//     Term 57 (AT2002-0250)/Term 58 (AT2002-5250)/FB Inputs/Value Channel 14 <-> Data Pointer/RawPositionValues[13]
//     Term 57 (AT2002-0250)/Term 58 (AT2002-5250)/FB Inputs/Value Channel 15 <-> Data Pointer/RawPositionValues[14]
//     Term 57 (AT2002-0250)/Term 58 (AT2002-5250)/FB Inputs/Value Channel 16 <-> Data Pointer/RawPositionValues[15]
//     Term 57 (AT2002-0250)/Term 58 (AT2002-5250)/FB Inputs/Value Channel 17 <-> Data Pointer/RawPositionValues[16]
//     Term 57 (AT2002-0250)/Term 58 (AT2002-5250)/FB Inputs/Value Channel 18 <-> Data Pointer/RawPositionValues[17]
//     Term 57 (AT2002-0250)/Term 58 (AT2002-5250)/FB Inputs/Value Channel 19 <-> Data Pointer/RawPositionValues[18]
//     Term 57 (AT2002-0250)/Term 58 (AT2002-5250)/FB Inputs/Value Channel 20 <-> Data Pointer/RawPositionValues[19]
//     Term 57 (AT2002-0250)/Term 58 (AT2002-5250)/FB Inputs/Value Channel 21 <-> Data Pointer/RawPositionValues[20]
//     Term 57 (AT2002-0250)/Term 58 (AT2002-5250)/FB Inputs/Value Channel 22 <-> Data Pointer/RawPositionValues[21]
//     Term 57 (AT2002-0250)/Term 58 (AT2002-5250)/FB Inputs/Value Channel 23 <-> Data Pointer/RawPositionValues[22]
//     Term 57 (AT2002-0250)/Term 58 (AT2002-5250)/FB Inputs/Value Channel 24 <-> Data Pointer/RawPositionValues[23]
//     Term 57 (AT2002-0250)/Term 58 (AT2002-5250)/FB Inputs/Value Channel 25 <-> Data Pointer/RawPositionValues[24]
//     Term 57 (AT2002-0250)/Term 58 (AT2002-5250)/FB Inputs/Value Channel 26 <-> Data Pointer/RawPositionValues[25]
//     Term 57 (AT2002-0250)/Term 58 (AT2002-5250)/FB Inputs/Value Channel 27 <-> Data Pointer/RawPositionValues[26]
//     Term 57 (AT2002-0250)/Term 58 (AT2002-5250)/FB Inputs/Value Channel 28 <-> Data Pointer/RawPositionValues[27]
//     Term 57 (AT2002-0250)/Term 58 (AT2002-5250)/FB Inputs/Value Channel 29 <-> Data Pointer/RawPositionValues[28]
//     Term 57 (AT2002-0250)/Term 58 (AT2002-5250)/FB Inputs/Value Channel 30 <-> Data Pointer/RawPositionValues[29]
//     Term 57 (AT2002-0250)/Term 58 (AT2002-5250)/FB Inputs/Value Channel 31 <-> Data Pointer/RawPositionValues[30]
//     Term 57 (AT2002-0250)/Term 58 (AT2002-5250)/FB Inputs/Value Channel 32 <-> Data Pointer/RawPositionValues[31]
//   Device 30 <-> TcCOM Objects/XTS ProcessingUnit 1/Part 1/Module 45
//     Term 59 (AT2200-0500)/CC Inputs/Current actual value Ch.1 <-> Data Pointer/CurrentActualValues[0]
//     Term 59 (AT2200-0500)/CC Inputs/Current actual value Ch.10 <-> Data Pointer/CurrentActualValues[9]
//     Term 59 (AT2200-0500)/CC Inputs/Current actual value Ch.11 <-> Data Pointer/CurrentActualValues[10]
//     Term 59 (AT2200-0500)/CC Inputs/Current actual value Ch.12 <-> Data Pointer/CurrentActualValues[11]
//     Term 59 (AT2200-0500)/CC Inputs/Current actual value Ch.13 <-> Data Pointer/CurrentActualValues[12]
//     Term 59 (AT2200-0500)/CC Inputs/Current actual value Ch.14 <-> Data Pointer/CurrentActualValues[13]
//     Term 59 (AT2200-0500)/CC Inputs/Current actual value Ch.15 <-> Data Pointer/CurrentActualValues[14]
//     Term 59 (AT2200-0500)/CC Inputs/Current actual value Ch.16 <-> Data Pointer/CurrentActualValues[15]
//     Term 59 (AT2200-0500)/CC Inputs/Current actual value Ch.17 <-> Data Pointer/CurrentActualValues[16]
//     Term 59 (AT2200-0500)/CC Inputs/Current actual value Ch.18 <-> Data Pointer/CurrentActualValues[17]
//     Term 59 (AT2200-0500)/CC Inputs/Current actual value Ch.19 <-> Data Pointer/CurrentActualValues[18]
//     Term 59 (AT2200-0500)/CC Inputs/Current actual value Ch.2 <-> Data Pointer/CurrentActualValues[1]
//     Term 59 (AT2200-0500)/CC Inputs/Current actual value Ch.20 <-> Data Pointer/CurrentActualValues[19]
//     Term 59 (AT2200-0500)/CC Inputs/Current actual value Ch.21 <-> Data Pointer/CurrentActualValues[20]
//     Term 59 (AT2200-0500)/CC Inputs/Current actual value Ch.22 <-> Data Pointer/CurrentActualValues[21]
//     Term 59 (AT2200-0500)/CC Inputs/Current actual value Ch.23 <-> Data Pointer/CurrentActualValues[22]
//     Term 59 (AT2200-0500)/CC Inputs/Current actual value Ch.24 <-> Data Pointer/CurrentActualValues[23]
//     Term 59 (AT2200-0500)/CC Inputs/Current actual value Ch.25 <-> Data Pointer/CurrentActualValues[24]
//     Term 59 (AT2200-0500)/CC Inputs/Current actual value Ch.26 <-> Data Pointer/CurrentActualValues[25]
//     Term 59 (AT2200-0500)/CC Inputs/Current actual value Ch.27 <-> Data Pointer/CurrentActualValues[26]
//     Term 59 (AT2200-0500)/CC Inputs/Current actual value Ch.28 <-> Data Pointer/CurrentActualValues[27]
//     Term 59 (AT2200-0500)/CC Inputs/Current actual value Ch.29 <-> Data Pointer/CurrentActualValues[28]
//     Term 59 (AT2200-0500)/CC Inputs/Current actual value Ch.3 <-> Data Pointer/CurrentActualValues[2]
//     Term 59 (AT2200-0500)/CC Inputs/Current actual value Ch.30 <-> Data Pointer/CurrentActualValues[29]
//     Term 59 (AT2200-0500)/CC Inputs/Current actual value Ch.4 <-> Data Pointer/CurrentActualValues[3]
//     Term 59 (AT2200-0500)/CC Inputs/Current actual value Ch.5 <-> Data Pointer/CurrentActualValues[4]
//     Term 59 (AT2200-0500)/CC Inputs/Current actual value Ch.6 <-> Data Pointer/CurrentActualValues[5]
//     Term 59 (AT2200-0500)/CC Inputs/Current actual value Ch.7 <-> Data Pointer/CurrentActualValues[6]
//     Term 59 (AT2200-0500)/CC Inputs/Current actual value Ch.8 <-> Data Pointer/CurrentActualValues[7]
//     Term 59 (AT2200-0500)/CC Inputs/Current actual value Ch.9 <-> Data Pointer/CurrentActualValues[8]
//     Term 59 (AT2200-0500)/CC Inputs/Status <-> Data Pointer/Status
//     Term 59 (AT2200-0500)/CC Outputs/Control <-> Data Pointer/Control
//     Term 59 (AT2200-0500)/CC Outputs/Current setpoint value Ch.1 <-> Data Pointer/CurrentSetpointValues[0]
//     Term 59 (AT2200-0500)/CC Outputs/Current setpoint value Ch.10 <-> Data Pointer/CurrentSetpointValues[9]
//     Term 59 (AT2200-0500)/CC Outputs/Current setpoint value Ch.11 <-> Data Pointer/CurrentSetpointValues[10]
//     Term 59 (AT2200-0500)/CC Outputs/Current setpoint value Ch.12 <-> Data Pointer/CurrentSetpointValues[11]
//     Term 59 (AT2200-0500)/CC Outputs/Current setpoint value Ch.13 <-> Data Pointer/CurrentSetpointValues[12]
//     Term 59 (AT2200-0500)/CC Outputs/Current setpoint value Ch.14 <-> Data Pointer/CurrentSetpointValues[13]
//     Term 59 (AT2200-0500)/CC Outputs/Current setpoint value Ch.15 <-> Data Pointer/CurrentSetpointValues[14]
//     Term 59 (AT2200-0500)/CC Outputs/Current setpoint value Ch.16 <-> Data Pointer/CurrentSetpointValues[15]
//     Term 59 (AT2200-0500)/CC Outputs/Current setpoint value Ch.17 <-> Data Pointer/CurrentSetpointValues[16]
//     Term 59 (AT2200-0500)/CC Outputs/Current setpoint value Ch.18 <-> Data Pointer/CurrentSetpointValues[17]
//     Term 59 (AT2200-0500)/CC Outputs/Current setpoint value Ch.19 <-> Data Pointer/CurrentSetpointValues[18]
//     Term 59 (AT2200-0500)/CC Outputs/Current setpoint value Ch.2 <-> Data Pointer/CurrentSetpointValues[1]
//     Term 59 (AT2200-0500)/CC Outputs/Current setpoint value Ch.20 <-> Data Pointer/CurrentSetpointValues[19]
//     Term 59 (AT2200-0500)/CC Outputs/Current setpoint value Ch.21 <-> Data Pointer/CurrentSetpointValues[20]
//     Term 59 (AT2200-0500)/CC Outputs/Current setpoint value Ch.22 <-> Data Pointer/CurrentSetpointValues[21]
//     Term 59 (AT2200-0500)/CC Outputs/Current setpoint value Ch.23 <-> Data Pointer/CurrentSetpointValues[22]
//     Term 59 (AT2200-0500)/CC Outputs/Current setpoint value Ch.24 <-> Data Pointer/CurrentSetpointValues[23]
//     Term 59 (AT2200-0500)/CC Outputs/Current setpoint value Ch.25 <-> Data Pointer/CurrentSetpointValues[24]
//     Term 59 (AT2200-0500)/CC Outputs/Current setpoint value Ch.26 <-> Data Pointer/CurrentSetpointValues[25]
//     Term 59 (AT2200-0500)/CC Outputs/Current setpoint value Ch.27 <-> Data Pointer/CurrentSetpointValues[26]
//     Term 59 (AT2200-0500)/CC Outputs/Current setpoint value Ch.28 <-> Data Pointer/CurrentSetpointValues[27]
//     Term 59 (AT2200-0500)/CC Outputs/Current setpoint value Ch.29 <-> Data Pointer/CurrentSetpointValues[28]
//     Term 59 (AT2200-0500)/CC Outputs/Current setpoint value Ch.3 <-> Data Pointer/CurrentSetpointValues[2]
//     Term 59 (AT2200-0500)/CC Outputs/Current setpoint value Ch.30 <-> Data Pointer/CurrentSetpointValues[29]
//     Term 59 (AT2200-0500)/CC Outputs/Current setpoint value Ch.4 <-> Data Pointer/CurrentSetpointValues[3]
//     Term 59 (AT2200-0500)/CC Outputs/Current setpoint value Ch.5 <-> Data Pointer/CurrentSetpointValues[4]
//     Term 59 (AT2200-0500)/CC Outputs/Current setpoint value Ch.6 <-> Data Pointer/CurrentSetpointValues[5]
//     Term 59 (AT2200-0500)/CC Outputs/Current setpoint value Ch.7 <-> Data Pointer/CurrentSetpointValues[6]
//     Term 59 (AT2200-0500)/CC Outputs/Current setpoint value Ch.8 <-> Data Pointer/CurrentSetpointValues[7]
//     Term 59 (AT2200-0500)/CC Outputs/Current setpoint value Ch.9 <-> Data Pointer/CurrentSetpointValues[8]
//     Term 59 (AT2200-0500)/LFB Inputs/BinaryData <-> Data Pointer/HallSensorValues
//   Device 30 <-> TcCOM Objects/XTS ProcessingUnit 1/Part 1/Module 46
//     Term 60 (AT2200-0500)/CC Inputs/Current actual value Ch.1 <-> Data Pointer/CurrentActualValues[0]
//     Term 60 (AT2200-0500)/CC Inputs/Current actual value Ch.10 <-> Data Pointer/CurrentActualValues[9]
//     Term 60 (AT2200-0500)/CC Inputs/Current actual value Ch.11 <-> Data Pointer/CurrentActualValues[10]
//     Term 60 (AT2200-0500)/CC Inputs/Current actual value Ch.12 <-> Data Pointer/CurrentActualValues[11]
//     Term 60 (AT2200-0500)/CC Inputs/Current actual value Ch.13 <-> Data Pointer/CurrentActualValues[12]
//     Term 60 (AT2200-0500)/CC Inputs/Current actual value Ch.14 <-> Data Pointer/CurrentActualValues[13]
//     Term 60 (AT2200-0500)/CC Inputs/Current actual value Ch.15 <-> Data Pointer/CurrentActualValues[14]
//     Term 60 (AT2200-0500)/CC Inputs/Current actual value Ch.16 <-> Data Pointer/CurrentActualValues[15]
//     Term 60 (AT2200-0500)/CC Inputs/Current actual value Ch.17 <-> Data Pointer/CurrentActualValues[16]
//     Term 60 (AT2200-0500)/CC Inputs/Current actual value Ch.18 <-> Data Pointer/CurrentActualValues[17]
//     Term 60 (AT2200-0500)/CC Inputs/Current actual value Ch.19 <-> Data Pointer/CurrentActualValues[18]
//     Term 60 (AT2200-0500)/CC Inputs/Current actual value Ch.2 <-> Data Pointer/CurrentActualValues[1]
//     Term 60 (AT2200-0500)/CC Inputs/Current actual value Ch.20 <-> Data Pointer/CurrentActualValues[19]
//     Term 60 (AT2200-0500)/CC Inputs/Current actual value Ch.21 <-> Data Pointer/CurrentActualValues[20]
//     Term 60 (AT2200-0500)/CC Inputs/Current actual value Ch.22 <-> Data Pointer/CurrentActualValues[21]
//     Term 60 (AT2200-0500)/CC Inputs/Current actual value Ch.23 <-> Data Pointer/CurrentActualValues[22]
//     Term 60 (AT2200-0500)/CC Inputs/Current actual value Ch.24 <-> Data Pointer/CurrentActualValues[23]
//     Term 60 (AT2200-0500)/CC Inputs/Current actual value Ch.25 <-> Data Pointer/CurrentActualValues[24]
//     Term 60 (AT2200-0500)/CC Inputs/Current actual value Ch.26 <-> Data Pointer/CurrentActualValues[25]
//     Term 60 (AT2200-0500)/CC Inputs/Current actual value Ch.27 <-> Data Pointer/CurrentActualValues[26]
//     Term 60 (AT2200-0500)/CC Inputs/Current actual value Ch.28 <-> Data Pointer/CurrentActualValues[27]
//     Term 60 (AT2200-0500)/CC Inputs/Current actual value Ch.29 <-> Data Pointer/CurrentActualValues[28]
//     Term 60 (AT2200-0500)/CC Inputs/Current actual value Ch.3 <-> Data Pointer/CurrentActualValues[2]
//     Term 60 (AT2200-0500)/CC Inputs/Current actual value Ch.30 <-> Data Pointer/CurrentActualValues[29]
//     Term 60 (AT2200-0500)/CC Inputs/Current actual value Ch.4 <-> Data Pointer/CurrentActualValues[3]
//     Term 60 (AT2200-0500)/CC Inputs/Current actual value Ch.5 <-> Data Pointer/CurrentActualValues[4]
//     Term 60 (AT2200-0500)/CC Inputs/Current actual value Ch.6 <-> Data Pointer/CurrentActualValues[5]
//     Term 60 (AT2200-0500)/CC Inputs/Current actual value Ch.7 <-> Data Pointer/CurrentActualValues[6]
//     Term 60 (AT2200-0500)/CC Inputs/Current actual value Ch.8 <-> Data Pointer/CurrentActualValues[7]
//     Term 60 (AT2200-0500)/CC Inputs/Current actual value Ch.9 <-> Data Pointer/CurrentActualValues[8]
//     Term 60 (AT2200-0500)/CC Inputs/Status <-> Data Pointer/Status
//     Term 60 (AT2200-0500)/CC Outputs/Control <-> Data Pointer/Control
//     Term 60 (AT2200-0500)/CC Outputs/Current setpoint value Ch.1 <-> Data Pointer/CurrentSetpointValues[0]
//     Term 60 (AT2200-0500)/CC Outputs/Current setpoint value Ch.10 <-> Data Pointer/CurrentSetpointValues[9]
//     Term 60 (AT2200-0500)/CC Outputs/Current setpoint value Ch.11 <-> Data Pointer/CurrentSetpointValues[10]
//     Term 60 (AT2200-0500)/CC Outputs/Current setpoint value Ch.12 <-> Data Pointer/CurrentSetpointValues[11]
//     Term 60 (AT2200-0500)/CC Outputs/Current setpoint value Ch.13 <-> Data Pointer/CurrentSetpointValues[12]
//     Term 60 (AT2200-0500)/CC Outputs/Current setpoint value Ch.14 <-> Data Pointer/CurrentSetpointValues[13]
//     Term 60 (AT2200-0500)/CC Outputs/Current setpoint value Ch.15 <-> Data Pointer/CurrentSetpointValues[14]
//     Term 60 (AT2200-0500)/CC Outputs/Current setpoint value Ch.16 <-> Data Pointer/CurrentSetpointValues[15]
//     Term 60 (AT2200-0500)/CC Outputs/Current setpoint value Ch.17 <-> Data Pointer/CurrentSetpointValues[16]
//     Term 60 (AT2200-0500)/CC Outputs/Current setpoint value Ch.18 <-> Data Pointer/CurrentSetpointValues[17]
//     Term 60 (AT2200-0500)/CC Outputs/Current setpoint value Ch.19 <-> Data Pointer/CurrentSetpointValues[18]
//     Term 60 (AT2200-0500)/CC Outputs/Current setpoint value Ch.2 <-> Data Pointer/CurrentSetpointValues[1]
//     Term 60 (AT2200-0500)/CC Outputs/Current setpoint value Ch.20 <-> Data Pointer/CurrentSetpointValues[19]
//     Term 60 (AT2200-0500)/CC Outputs/Current setpoint value Ch.21 <-> Data Pointer/CurrentSetpointValues[20]
//     Term 60 (AT2200-0500)/CC Outputs/Current setpoint value Ch.22 <-> Data Pointer/CurrentSetpointValues[21]
//     Term 60 (AT2200-0500)/CC Outputs/Current setpoint value Ch.23 <-> Data Pointer/CurrentSetpointValues[22]
//     Term 60 (AT2200-0500)/CC Outputs/Current setpoint value Ch.24 <-> Data Pointer/CurrentSetpointValues[23]
//     Term 60 (AT2200-0500)/CC Outputs/Current setpoint value Ch.25 <-> Data Pointer/CurrentSetpointValues[24]
//     Term 60 (AT2200-0500)/CC Outputs/Current setpoint value Ch.26 <-> Data Pointer/CurrentSetpointValues[25]
//     Term 60 (AT2200-0500)/CC Outputs/Current setpoint value Ch.27 <-> Data Pointer/CurrentSetpointValues[26]
//     Term 60 (AT2200-0500)/CC Outputs/Current setpoint value Ch.28 <-> Data Pointer/CurrentSetpointValues[27]
//     Term 60 (AT2200-0500)/CC Outputs/Current setpoint value Ch.29 <-> Data Pointer/CurrentSetpointValues[28]
//     Term 60 (AT2200-0500)/CC Outputs/Current setpoint value Ch.3 <-> Data Pointer/CurrentSetpointValues[2]
//     Term 60 (AT2200-0500)/CC Outputs/Current setpoint value Ch.30 <-> Data Pointer/CurrentSetpointValues[29]
//     Term 60 (AT2200-0500)/CC Outputs/Current setpoint value Ch.4 <-> Data Pointer/CurrentSetpointValues[3]
//     Term 60 (AT2200-0500)/CC Outputs/Current setpoint value Ch.5 <-> Data Pointer/CurrentSetpointValues[4]
//     Term 60 (AT2200-0500)/CC Outputs/Current setpoint value Ch.6 <-> Data Pointer/CurrentSetpointValues[5]
//     Term 60 (AT2200-0500)/CC Outputs/Current setpoint value Ch.7 <-> Data Pointer/CurrentSetpointValues[6]
//     Term 60 (AT2200-0500)/CC Outputs/Current setpoint value Ch.8 <-> Data Pointer/CurrentSetpointValues[7]
//     Term 60 (AT2200-0500)/CC Outputs/Current setpoint value Ch.9 <-> Data Pointer/CurrentSetpointValues[8]
//     Term 60 (AT2200-0500)/LFB Inputs/BinaryData <-> Data Pointer/HallSensorValues
//   Device 31 <-> TcCOM Objects/XTS ProcessingUnit 1/Part 1/Module 47
//     Term 61 (AT2202-0500)/CC Inputs/Current actual value Ch.1 <-> Data Pointer/CurrentActualValues[0]
//     Term 61 (AT2202-0500)/CC Inputs/Current actual value Ch.10 <-> Data Pointer/CurrentActualValues[9]
//     Term 61 (AT2202-0500)/CC Inputs/Current actual value Ch.11 <-> Data Pointer/CurrentActualValues[10]
//     Term 61 (AT2202-0500)/CC Inputs/Current actual value Ch.12 <-> Data Pointer/CurrentActualValues[11]
//     Term 61 (AT2202-0500)/CC Inputs/Current actual value Ch.13 <-> Data Pointer/CurrentActualValues[12]
//     Term 61 (AT2202-0500)/CC Inputs/Current actual value Ch.14 <-> Data Pointer/CurrentActualValues[13]
//     Term 61 (AT2202-0500)/CC Inputs/Current actual value Ch.15 <-> Data Pointer/CurrentActualValues[14]
//     Term 61 (AT2202-0500)/CC Inputs/Current actual value Ch.16 <-> Data Pointer/CurrentActualValues[15]
//     Term 61 (AT2202-0500)/CC Inputs/Current actual value Ch.17 <-> Data Pointer/CurrentActualValues[16]
//     Term 61 (AT2202-0500)/CC Inputs/Current actual value Ch.18 <-> Data Pointer/CurrentActualValues[17]
//     Term 61 (AT2202-0500)/CC Inputs/Current actual value Ch.19 <-> Data Pointer/CurrentActualValues[18]
//     Term 61 (AT2202-0500)/CC Inputs/Current actual value Ch.2 <-> Data Pointer/CurrentActualValues[1]
//     Term 61 (AT2202-0500)/CC Inputs/Current actual value Ch.20 <-> Data Pointer/CurrentActualValues[19]
//     Term 61 (AT2202-0500)/CC Inputs/Current actual value Ch.21 <-> Data Pointer/CurrentActualValues[20]
//     Term 61 (AT2202-0500)/CC Inputs/Current actual value Ch.22 <-> Data Pointer/CurrentActualValues[21]
//     Term 61 (AT2202-0500)/CC Inputs/Current actual value Ch.23 <-> Data Pointer/CurrentActualValues[22]
//     Term 61 (AT2202-0500)/CC Inputs/Current actual value Ch.24 <-> Data Pointer/CurrentActualValues[23]
//     Term 61 (AT2202-0500)/CC Inputs/Current actual value Ch.25 <-> Data Pointer/CurrentActualValues[24]
//     Term 61 (AT2202-0500)/CC Inputs/Current actual value Ch.26 <-> Data Pointer/CurrentActualValues[25]
//     Term 61 (AT2202-0500)/CC Inputs/Current actual value Ch.27 <-> Data Pointer/CurrentActualValues[26]
//     Term 61 (AT2202-0500)/CC Inputs/Current actual value Ch.28 <-> Data Pointer/CurrentActualValues[27]
//     Term 61 (AT2202-0500)/CC Inputs/Current actual value Ch.29 <-> Data Pointer/CurrentActualValues[28]
//     Term 61 (AT2202-0500)/CC Inputs/Current actual value Ch.3 <-> Data Pointer/CurrentActualValues[2]
//     Term 61 (AT2202-0500)/CC Inputs/Current actual value Ch.30 <-> Data Pointer/CurrentActualValues[29]
//     Term 61 (AT2202-0500)/CC Inputs/Current actual value Ch.4 <-> Data Pointer/CurrentActualValues[3]
//     Term 61 (AT2202-0500)/CC Inputs/Current actual value Ch.5 <-> Data Pointer/CurrentActualValues[4]
//     Term 61 (AT2202-0500)/CC Inputs/Current actual value Ch.6 <-> Data Pointer/CurrentActualValues[5]
//     Term 61 (AT2202-0500)/CC Inputs/Current actual value Ch.7 <-> Data Pointer/CurrentActualValues[6]
//     Term 61 (AT2202-0500)/CC Inputs/Current actual value Ch.8 <-> Data Pointer/CurrentActualValues[7]
//     Term 61 (AT2202-0500)/CC Inputs/Current actual value Ch.9 <-> Data Pointer/CurrentActualValues[8]
//     Term 61 (AT2202-0500)/CC Inputs/Status <-> Data Pointer/Status
//     Term 61 (AT2202-0500)/CC Outputs/Control <-> Data Pointer/Control
//     Term 61 (AT2202-0500)/CC Outputs/Current setpoint value Ch.1 <-> Data Pointer/CurrentSetpointValues[0]
//     Term 61 (AT2202-0500)/CC Outputs/Current setpoint value Ch.10 <-> Data Pointer/CurrentSetpointValues[9]
//     Term 61 (AT2202-0500)/CC Outputs/Current setpoint value Ch.11 <-> Data Pointer/CurrentSetpointValues[10]
//     Term 61 (AT2202-0500)/CC Outputs/Current setpoint value Ch.12 <-> Data Pointer/CurrentSetpointValues[11]
//     Term 61 (AT2202-0500)/CC Outputs/Current setpoint value Ch.13 <-> Data Pointer/CurrentSetpointValues[12]
//     Term 61 (AT2202-0500)/CC Outputs/Current setpoint value Ch.14 <-> Data Pointer/CurrentSetpointValues[13]
//     Term 61 (AT2202-0500)/CC Outputs/Current setpoint value Ch.15 <-> Data Pointer/CurrentSetpointValues[14]
//     Term 61 (AT2202-0500)/CC Outputs/Current setpoint value Ch.16 <-> Data Pointer/CurrentSetpointValues[15]
//     Term 61 (AT2202-0500)/CC Outputs/Current setpoint value Ch.17 <-> Data Pointer/CurrentSetpointValues[16]
//     Term 61 (AT2202-0500)/CC Outputs/Current setpoint value Ch.18 <-> Data Pointer/CurrentSetpointValues[17]
//     Term 61 (AT2202-0500)/CC Outputs/Current setpoint value Ch.19 <-> Data Pointer/CurrentSetpointValues[18]
//     Term 61 (AT2202-0500)/CC Outputs/Current setpoint value Ch.2 <-> Data Pointer/CurrentSetpointValues[1]
//     Term 61 (AT2202-0500)/CC Outputs/Current setpoint value Ch.20 <-> Data Pointer/CurrentSetpointValues[19]
//     Term 61 (AT2202-0500)/CC Outputs/Current setpoint value Ch.21 <-> Data Pointer/CurrentSetpointValues[20]
//     Term 61 (AT2202-0500)/CC Outputs/Current setpoint value Ch.22 <-> Data Pointer/CurrentSetpointValues[21]
//     Term 61 (AT2202-0500)/CC Outputs/Current setpoint value Ch.23 <-> Data Pointer/CurrentSetpointValues[22]
//     Term 61 (AT2202-0500)/CC Outputs/Current setpoint value Ch.24 <-> Data Pointer/CurrentSetpointValues[23]
//     Term 61 (AT2202-0500)/CC Outputs/Current setpoint value Ch.25 <-> Data Pointer/CurrentSetpointValues[24]
//     Term 61 (AT2202-0500)/CC Outputs/Current setpoint value Ch.26 <-> Data Pointer/CurrentSetpointValues[25]
//     Term 61 (AT2202-0500)/CC Outputs/Current setpoint value Ch.27 <-> Data Pointer/CurrentSetpointValues[26]
//     Term 61 (AT2202-0500)/CC Outputs/Current setpoint value Ch.28 <-> Data Pointer/CurrentSetpointValues[27]
//     Term 61 (AT2202-0500)/CC Outputs/Current setpoint value Ch.29 <-> Data Pointer/CurrentSetpointValues[28]
//     Term 61 (AT2202-0500)/CC Outputs/Current setpoint value Ch.3 <-> Data Pointer/CurrentSetpointValues[2]
//     Term 61 (AT2202-0500)/CC Outputs/Current setpoint value Ch.30 <-> Data Pointer/CurrentSetpointValues[29]
//     Term 61 (AT2202-0500)/CC Outputs/Current setpoint value Ch.4 <-> Data Pointer/CurrentSetpointValues[3]
//     Term 61 (AT2202-0500)/CC Outputs/Current setpoint value Ch.5 <-> Data Pointer/CurrentSetpointValues[4]
//     Term 61 (AT2202-0500)/CC Outputs/Current setpoint value Ch.6 <-> Data Pointer/CurrentSetpointValues[5]
//     Term 61 (AT2202-0500)/CC Outputs/Current setpoint value Ch.7 <-> Data Pointer/CurrentSetpointValues[6]
//     Term 61 (AT2202-0500)/CC Outputs/Current setpoint value Ch.8 <-> Data Pointer/CurrentSetpointValues[7]
//     Term 61 (AT2202-0500)/CC Outputs/Current setpoint value Ch.9 <-> Data Pointer/CurrentSetpointValues[8]
//     Term 61 (AT2202-0500)/LFB Inputs/BinaryData <-> Data Pointer/HallSensorValues
//   Device 31 <-> TcCOM Objects/XTS ProcessingUnit 1/Part 1/Module 48
//     Term 62 (AT2200-0500)/CC Inputs/Current actual value Ch.1 <-> Data Pointer/CurrentActualValues[0]
//     Term 62 (AT2200-0500)/CC Inputs/Current actual value Ch.10 <-> Data Pointer/CurrentActualValues[9]
//     Term 62 (AT2200-0500)/CC Inputs/Current actual value Ch.11 <-> Data Pointer/CurrentActualValues[10]
//     Term 62 (AT2200-0500)/CC Inputs/Current actual value Ch.12 <-> Data Pointer/CurrentActualValues[11]
//     Term 62 (AT2200-0500)/CC Inputs/Current actual value Ch.13 <-> Data Pointer/CurrentActualValues[12]
//     Term 62 (AT2200-0500)/CC Inputs/Current actual value Ch.14 <-> Data Pointer/CurrentActualValues[13]
//     Term 62 (AT2200-0500)/CC Inputs/Current actual value Ch.15 <-> Data Pointer/CurrentActualValues[14]
//     Term 62 (AT2200-0500)/CC Inputs/Current actual value Ch.16 <-> Data Pointer/CurrentActualValues[15]
//     Term 62 (AT2200-0500)/CC Inputs/Current actual value Ch.17 <-> Data Pointer/CurrentActualValues[16]
//     Term 62 (AT2200-0500)/CC Inputs/Current actual value Ch.18 <-> Data Pointer/CurrentActualValues[17]
//     Term 62 (AT2200-0500)/CC Inputs/Current actual value Ch.19 <-> Data Pointer/CurrentActualValues[18]
//     Term 62 (AT2200-0500)/CC Inputs/Current actual value Ch.2 <-> Data Pointer/CurrentActualValues[1]
//     Term 62 (AT2200-0500)/CC Inputs/Current actual value Ch.20 <-> Data Pointer/CurrentActualValues[19]
//     Term 62 (AT2200-0500)/CC Inputs/Current actual value Ch.21 <-> Data Pointer/CurrentActualValues[20]
//     Term 62 (AT2200-0500)/CC Inputs/Current actual value Ch.22 <-> Data Pointer/CurrentActualValues[21]
//     Term 62 (AT2200-0500)/CC Inputs/Current actual value Ch.23 <-> Data Pointer/CurrentActualValues[22]
//     Term 62 (AT2200-0500)/CC Inputs/Current actual value Ch.24 <-> Data Pointer/CurrentActualValues[23]
//     Term 62 (AT2200-0500)/CC Inputs/Current actual value Ch.25 <-> Data Pointer/CurrentActualValues[24]
//     Term 62 (AT2200-0500)/CC Inputs/Current actual value Ch.26 <-> Data Pointer/CurrentActualValues[25]
//     Term 62 (AT2200-0500)/CC Inputs/Current actual value Ch.27 <-> Data Pointer/CurrentActualValues[26]
//     Term 62 (AT2200-0500)/CC Inputs/Current actual value Ch.28 <-> Data Pointer/CurrentActualValues[27]
//     Term 62 (AT2200-0500)/CC Inputs/Current actual value Ch.29 <-> Data Pointer/CurrentActualValues[28]
//     Term 62 (AT2200-0500)/CC Inputs/Current actual value Ch.3 <-> Data Pointer/CurrentActualValues[2]
//     Term 62 (AT2200-0500)/CC Inputs/Current actual value Ch.30 <-> Data Pointer/CurrentActualValues[29]
//     Term 62 (AT2200-0500)/CC Inputs/Current actual value Ch.4 <-> Data Pointer/CurrentActualValues[3]
//     Term 62 (AT2200-0500)/CC Inputs/Current actual value Ch.5 <-> Data Pointer/CurrentActualValues[4]
//     Term 62 (AT2200-0500)/CC Inputs/Current actual value Ch.6 <-> Data Pointer/CurrentActualValues[5]
//     Term 62 (AT2200-0500)/CC Inputs/Current actual value Ch.7 <-> Data Pointer/CurrentActualValues[6]
//     Term 62 (AT2200-0500)/CC Inputs/Current actual value Ch.8 <-> Data Pointer/CurrentActualValues[7]
//     Term 62 (AT2200-0500)/CC Inputs/Current actual value Ch.9 <-> Data Pointer/CurrentActualValues[8]
//     Term 62 (AT2200-0500)/CC Inputs/Status <-> Data Pointer/Status
//     Term 62 (AT2200-0500)/CC Outputs/Control <-> Data Pointer/Control
//     Term 62 (AT2200-0500)/CC Outputs/Current setpoint value Ch.1 <-> Data Pointer/CurrentSetpointValues[0]
//     Term 62 (AT2200-0500)/CC Outputs/Current setpoint value Ch.10 <-> Data Pointer/CurrentSetpointValues[9]
//     Term 62 (AT2200-0500)/CC Outputs/Current setpoint value Ch.11 <-> Data Pointer/CurrentSetpointValues[10]
//     Term 62 (AT2200-0500)/CC Outputs/Current setpoint value Ch.12 <-> Data Pointer/CurrentSetpointValues[11]
//     Term 62 (AT2200-0500)/CC Outputs/Current setpoint value Ch.13 <-> Data Pointer/CurrentSetpointValues[12]
//     Term 62 (AT2200-0500)/CC Outputs/Current setpoint value Ch.14 <-> Data Pointer/CurrentSetpointValues[13]
//     Term 62 (AT2200-0500)/CC Outputs/Current setpoint value Ch.15 <-> Data Pointer/CurrentSetpointValues[14]
//     Term 62 (AT2200-0500)/CC Outputs/Current setpoint value Ch.16 <-> Data Pointer/CurrentSetpointValues[15]
//     Term 62 (AT2200-0500)/CC Outputs/Current setpoint value Ch.17 <-> Data Pointer/CurrentSetpointValues[16]
//     Term 62 (AT2200-0500)/CC Outputs/Current setpoint value Ch.18 <-> Data Pointer/CurrentSetpointValues[17]
//     Term 62 (AT2200-0500)/CC Outputs/Current setpoint value Ch.19 <-> Data Pointer/CurrentSetpointValues[18]
//     Term 62 (AT2200-0500)/CC Outputs/Current setpoint value Ch.2 <-> Data Pointer/CurrentSetpointValues[1]
//     Term 62 (AT2200-0500)/CC Outputs/Current setpoint value Ch.20 <-> Data Pointer/CurrentSetpointValues[19]
//     Term 62 (AT2200-0500)/CC Outputs/Current setpoint value Ch.21 <-> Data Pointer/CurrentSetpointValues[20]
//     Term 62 (AT2200-0500)/CC Outputs/Current setpoint value Ch.22 <-> Data Pointer/CurrentSetpointValues[21]
//     Term 62 (AT2200-0500)/CC Outputs/Current setpoint value Ch.23 <-> Data Pointer/CurrentSetpointValues[22]
//     Term 62 (AT2200-0500)/CC Outputs/Current setpoint value Ch.24 <-> Data Pointer/CurrentSetpointValues[23]
//     Term 62 (AT2200-0500)/CC Outputs/Current setpoint value Ch.25 <-> Data Pointer/CurrentSetpointValues[24]
//     Term 62 (AT2200-0500)/CC Outputs/Current setpoint value Ch.26 <-> Data Pointer/CurrentSetpointValues[25]
//     Term 62 (AT2200-0500)/CC Outputs/Current setpoint value Ch.27 <-> Data Pointer/CurrentSetpointValues[26]
//     Term 62 (AT2200-0500)/CC Outputs/Current setpoint value Ch.28 <-> Data Pointer/CurrentSetpointValues[27]
//     Term 62 (AT2200-0500)/CC Outputs/Current setpoint value Ch.29 <-> Data Pointer/CurrentSetpointValues[28]
//     Term 62 (AT2200-0500)/CC Outputs/Current setpoint value Ch.3 <-> Data Pointer/CurrentSetpointValues[2]
//     Term 62 (AT2200-0500)/CC Outputs/Current setpoint value Ch.30 <-> Data Pointer/CurrentSetpointValues[29]
//     Term 62 (AT2200-0500)/CC Outputs/Current setpoint value Ch.4 <-> Data Pointer/CurrentSetpointValues[3]
//     Term 62 (AT2200-0500)/CC Outputs/Current setpoint value Ch.5 <-> Data Pointer/CurrentSetpointValues[4]
//     Term 62 (AT2200-0500)/CC Outputs/Current setpoint value Ch.6 <-> Data Pointer/CurrentSetpointValues[5]
//     Term 62 (AT2200-0500)/CC Outputs/Current setpoint value Ch.7 <-> Data Pointer/CurrentSetpointValues[6]
//     Term 62 (AT2200-0500)/CC Outputs/Current setpoint value Ch.8 <-> Data Pointer/CurrentSetpointValues[7]
//     Term 62 (AT2200-0500)/CC Outputs/Current setpoint value Ch.9 <-> Data Pointer/CurrentSetpointValues[8]
//     Term 62 (AT2200-0500)/LFB Inputs/BinaryData <-> Data Pointer/HallSensorValues
//   Device 31 <-> TcCOM Objects/XTS ProcessingUnit 1/Part 1/Module 49
//     Term 63 (AT2000-0250)/CC Inputs/Current actual value Ch.1 <-> Data Pointer/CurrentActualValues[0]
//     Term 63 (AT2000-0250)/CC Inputs/Current actual value Ch.10 <-> Data Pointer/CurrentActualValues[9]
//     Term 63 (AT2000-0250)/CC Inputs/Current actual value Ch.11 <-> Data Pointer/CurrentActualValues[10]
//     Term 63 (AT2000-0250)/CC Inputs/Current actual value Ch.12 <-> Data Pointer/CurrentActualValues[11]
//     Term 63 (AT2000-0250)/CC Inputs/Current actual value Ch.13 <-> Data Pointer/CurrentActualValues[12]
//     Term 63 (AT2000-0250)/CC Inputs/Current actual value Ch.14 <-> Data Pointer/CurrentActualValues[13]
//     Term 63 (AT2000-0250)/CC Inputs/Current actual value Ch.15 <-> Data Pointer/CurrentActualValues[14]
//     Term 63 (AT2000-0250)/CC Inputs/Current actual value Ch.2 <-> Data Pointer/CurrentActualValues[1]
//     Term 63 (AT2000-0250)/CC Inputs/Current actual value Ch.3 <-> Data Pointer/CurrentActualValues[2]
//     Term 63 (AT2000-0250)/CC Inputs/Current actual value Ch.4 <-> Data Pointer/CurrentActualValues[3]
//     Term 63 (AT2000-0250)/CC Inputs/Current actual value Ch.5 <-> Data Pointer/CurrentActualValues[4]
//     Term 63 (AT2000-0250)/CC Inputs/Current actual value Ch.6 <-> Data Pointer/CurrentActualValues[5]
//     Term 63 (AT2000-0250)/CC Inputs/Current actual value Ch.7 <-> Data Pointer/CurrentActualValues[6]
//     Term 63 (AT2000-0250)/CC Inputs/Current actual value Ch.8 <-> Data Pointer/CurrentActualValues[7]
//     Term 63 (AT2000-0250)/CC Inputs/Current actual value Ch.9 <-> Data Pointer/CurrentActualValues[8]
//     Term 63 (AT2000-0250)/CC Inputs/Status <-> Data Pointer/Status
//     Term 63 (AT2000-0250)/CC Outputs/Control <-> Data Pointer/Control
//     Term 63 (AT2000-0250)/CC Outputs/Current setpoint value Ch.1 <-> Data Pointer/CurrentSetpointValues[0]
//     Term 63 (AT2000-0250)/CC Outputs/Current setpoint value Ch.10 <-> Data Pointer/CurrentSetpointValues[9]
//     Term 63 (AT2000-0250)/CC Outputs/Current setpoint value Ch.11 <-> Data Pointer/CurrentSetpointValues[10]
//     Term 63 (AT2000-0250)/CC Outputs/Current setpoint value Ch.12 <-> Data Pointer/CurrentSetpointValues[11]
//     Term 63 (AT2000-0250)/CC Outputs/Current setpoint value Ch.13 <-> Data Pointer/CurrentSetpointValues[12]
//     Term 63 (AT2000-0250)/CC Outputs/Current setpoint value Ch.14 <-> Data Pointer/CurrentSetpointValues[13]
//     Term 63 (AT2000-0250)/CC Outputs/Current setpoint value Ch.15 <-> Data Pointer/CurrentSetpointValues[14]
//     Term 63 (AT2000-0250)/CC Outputs/Current setpoint value Ch.2 <-> Data Pointer/CurrentSetpointValues[1]
//     Term 63 (AT2000-0250)/CC Outputs/Current setpoint value Ch.3 <-> Data Pointer/CurrentSetpointValues[2]
//     Term 63 (AT2000-0250)/CC Outputs/Current setpoint value Ch.4 <-> Data Pointer/CurrentSetpointValues[3]
//     Term 63 (AT2000-0250)/CC Outputs/Current setpoint value Ch.5 <-> Data Pointer/CurrentSetpointValues[4]
//     Term 63 (AT2000-0250)/CC Outputs/Current setpoint value Ch.6 <-> Data Pointer/CurrentSetpointValues[5]
//     Term 63 (AT2000-0250)/CC Outputs/Current setpoint value Ch.7 <-> Data Pointer/CurrentSetpointValues[6]
//     Term 63 (AT2000-0250)/CC Outputs/Current setpoint value Ch.8 <-> Data Pointer/CurrentSetpointValues[7]
//     Term 63 (AT2000-0250)/CC Outputs/Current setpoint value Ch.9 <-> Data Pointer/CurrentSetpointValues[8]
//     Term 63 (AT2000-0250)/Term 64 (AT2000-5250)/FB Inputs/Value Channel 01 <-> Data Pointer/RawPositionValues[0]
//     Term 63 (AT2000-0250)/Term 64 (AT2000-5250)/FB Inputs/Value Channel 02 <-> Data Pointer/RawPositionValues[1]
//     Term 63 (AT2000-0250)/Term 64 (AT2000-5250)/FB Inputs/Value Channel 03 <-> Data Pointer/RawPositionValues[2]
//     Term 63 (AT2000-0250)/Term 64 (AT2000-5250)/FB Inputs/Value Channel 04 <-> Data Pointer/RawPositionValues[3]
//     Term 63 (AT2000-0250)/Term 64 (AT2000-5250)/FB Inputs/Value Channel 05 <-> Data Pointer/RawPositionValues[4]
//     Term 63 (AT2000-0250)/Term 64 (AT2000-5250)/FB Inputs/Value Channel 06 <-> Data Pointer/RawPositionValues[5]
//     Term 63 (AT2000-0250)/Term 64 (AT2000-5250)/FB Inputs/Value Channel 07 <-> Data Pointer/RawPositionValues[6]
//     Term 63 (AT2000-0250)/Term 64 (AT2000-5250)/FB Inputs/Value Channel 08 <-> Data Pointer/RawPositionValues[7]
//     Term 63 (AT2000-0250)/Term 64 (AT2000-5250)/FB Inputs/Value Channel 09 <-> Data Pointer/RawPositionValues[8]
//     Term 63 (AT2000-0250)/Term 64 (AT2000-5250)/FB Inputs/Value Channel 10 <-> Data Pointer/RawPositionValues[9]
//     Term 63 (AT2000-0250)/Term 64 (AT2000-5250)/FB Inputs/Value Channel 11 <-> Data Pointer/RawPositionValues[10]
//     Term 63 (AT2000-0250)/Term 64 (AT2000-5250)/FB Inputs/Value Channel 12 <-> Data Pointer/RawPositionValues[11]
//     Term 63 (AT2000-0250)/Term 64 (AT2000-5250)/FB Inputs/Value Channel 13 <-> Data Pointer/RawPositionValues[12]
//     Term 63 (AT2000-0250)/Term 64 (AT2000-5250)/FB Inputs/Value Channel 14 <-> Data Pointer/RawPositionValues[13]
//     Term 63 (AT2000-0250)/Term 64 (AT2000-5250)/FB Inputs/Value Channel 15 <-> Data Pointer/RawPositionValues[14]
//     Term 63 (AT2000-0250)/Term 64 (AT2000-5250)/FB Inputs/Value Channel 16 <-> Data Pointer/RawPositionValues[15]
//     Term 63 (AT2000-0250)/Term 64 (AT2000-5250)/FB Inputs/Value Channel 17 <-> Data Pointer/RawPositionValues[16]
//     Term 63 (AT2000-0250)/Term 64 (AT2000-5250)/FB Inputs/Value Channel 18 <-> Data Pointer/RawPositionValues[17]
//     Term 63 (AT2000-0250)/Term 64 (AT2000-5250)/FB Inputs/Value Channel 19 <-> Data Pointer/RawPositionValues[18]
//     Term 63 (AT2000-0250)/Term 64 (AT2000-5250)/FB Inputs/Value Channel 20 <-> Data Pointer/RawPositionValues[19]
//     Term 63 (AT2000-0250)/Term 64 (AT2000-5250)/FB Inputs/Value Channel 21 <-> Data Pointer/RawPositionValues[20]
//     Term 63 (AT2000-0250)/Term 64 (AT2000-5250)/FB Inputs/Value Channel 22 <-> Data Pointer/RawPositionValues[21]
//     Term 63 (AT2000-0250)/Term 64 (AT2000-5250)/FB Inputs/Value Channel 23 <-> Data Pointer/RawPositionValues[22]
//     Term 63 (AT2000-0250)/Term 64 (AT2000-5250)/FB Inputs/Value Channel 24 <-> Data Pointer/RawPositionValues[23]
//     Term 63 (AT2000-0250)/Term 64 (AT2000-5250)/FB Inputs/Value Channel 25 <-> Data Pointer/RawPositionValues[24]
//     Term 63 (AT2000-0250)/Term 64 (AT2000-5250)/FB Inputs/Value Channel 26 <-> Data Pointer/RawPositionValues[25]
//     Term 63 (AT2000-0250)/Term 64 (AT2000-5250)/FB Inputs/Value Channel 27 <-> Data Pointer/RawPositionValues[26]
//     Term 63 (AT2000-0250)/Term 64 (AT2000-5250)/FB Inputs/Value Channel 28 <-> Data Pointer/RawPositionValues[27]
//     Term 63 (AT2000-0250)/Term 64 (AT2000-5250)/FB Inputs/Value Channel 29 <-> Data Pointer/RawPositionValues[28]
//     Term 63 (AT2000-0250)/Term 64 (AT2000-5250)/FB Inputs/Value Channel 30 <-> Data Pointer/RawPositionValues[29]
//     Term 63 (AT2000-0250)/Term 64 (AT2000-5250)/FB Inputs/Value Channel 31 <-> Data Pointer/RawPositionValues[30]
//     Term 63 (AT2000-0250)/Term 64 (AT2000-5250)/FB Inputs/Value Channel 32 <-> Data Pointer/RawPositionValues[31]
//   Device 32 <-> TcCOM Objects/XTS ProcessingUnit 1/Part 1/Module 50
//     Term 65 (AT2002-0250)/CC Inputs/Current actual value Ch.1 <-> Data Pointer/CurrentActualValues[0]
//     Term 65 (AT2002-0250)/CC Inputs/Current actual value Ch.10 <-> Data Pointer/CurrentActualValues[9]
//     Term 65 (AT2002-0250)/CC Inputs/Current actual value Ch.11 <-> Data Pointer/CurrentActualValues[10]
//     Term 65 (AT2002-0250)/CC Inputs/Current actual value Ch.12 <-> Data Pointer/CurrentActualValues[11]
//     Term 65 (AT2002-0250)/CC Inputs/Current actual value Ch.13 <-> Data Pointer/CurrentActualValues[12]
//     Term 65 (AT2002-0250)/CC Inputs/Current actual value Ch.14 <-> Data Pointer/CurrentActualValues[13]
//     Term 65 (AT2002-0250)/CC Inputs/Current actual value Ch.15 <-> Data Pointer/CurrentActualValues[14]
//     Term 65 (AT2002-0250)/CC Inputs/Current actual value Ch.2 <-> Data Pointer/CurrentActualValues[1]
//     Term 65 (AT2002-0250)/CC Inputs/Current actual value Ch.3 <-> Data Pointer/CurrentActualValues[2]
//     Term 65 (AT2002-0250)/CC Inputs/Current actual value Ch.4 <-> Data Pointer/CurrentActualValues[3]
//     Term 65 (AT2002-0250)/CC Inputs/Current actual value Ch.5 <-> Data Pointer/CurrentActualValues[4]
//     Term 65 (AT2002-0250)/CC Inputs/Current actual value Ch.6 <-> Data Pointer/CurrentActualValues[5]
//     Term 65 (AT2002-0250)/CC Inputs/Current actual value Ch.7 <-> Data Pointer/CurrentActualValues[6]
//     Term 65 (AT2002-0250)/CC Inputs/Current actual value Ch.8 <-> Data Pointer/CurrentActualValues[7]
//     Term 65 (AT2002-0250)/CC Inputs/Current actual value Ch.9 <-> Data Pointer/CurrentActualValues[8]
//     Term 65 (AT2002-0250)/CC Inputs/Status <-> Data Pointer/Status
//     Term 65 (AT2002-0250)/CC Outputs/Control <-> Data Pointer/Control
//     Term 65 (AT2002-0250)/CC Outputs/Current setpoint value Ch.1 <-> Data Pointer/CurrentSetpointValues[0]
//     Term 65 (AT2002-0250)/CC Outputs/Current setpoint value Ch.10 <-> Data Pointer/CurrentSetpointValues[9]
//     Term 65 (AT2002-0250)/CC Outputs/Current setpoint value Ch.11 <-> Data Pointer/CurrentSetpointValues[10]
//     Term 65 (AT2002-0250)/CC Outputs/Current setpoint value Ch.12 <-> Data Pointer/CurrentSetpointValues[11]
//     Term 65 (AT2002-0250)/CC Outputs/Current setpoint value Ch.13 <-> Data Pointer/CurrentSetpointValues[12]
//     Term 65 (AT2002-0250)/CC Outputs/Current setpoint value Ch.14 <-> Data Pointer/CurrentSetpointValues[13]
//     Term 65 (AT2002-0250)/CC Outputs/Current setpoint value Ch.15 <-> Data Pointer/CurrentSetpointValues[14]
//     Term 65 (AT2002-0250)/CC Outputs/Current setpoint value Ch.2 <-> Data Pointer/CurrentSetpointValues[1]
//     Term 65 (AT2002-0250)/CC Outputs/Current setpoint value Ch.3 <-> Data Pointer/CurrentSetpointValues[2]
//     Term 65 (AT2002-0250)/CC Outputs/Current setpoint value Ch.4 <-> Data Pointer/CurrentSetpointValues[3]
//     Term 65 (AT2002-0250)/CC Outputs/Current setpoint value Ch.5 <-> Data Pointer/CurrentSetpointValues[4]
//     Term 65 (AT2002-0250)/CC Outputs/Current setpoint value Ch.6 <-> Data Pointer/CurrentSetpointValues[5]
//     Term 65 (AT2002-0250)/CC Outputs/Current setpoint value Ch.7 <-> Data Pointer/CurrentSetpointValues[6]
//     Term 65 (AT2002-0250)/CC Outputs/Current setpoint value Ch.8 <-> Data Pointer/CurrentSetpointValues[7]
//     Term 65 (AT2002-0250)/CC Outputs/Current setpoint value Ch.9 <-> Data Pointer/CurrentSetpointValues[8]
//     Term 65 (AT2002-0250)/Term 66 (AT2002-5250)/FB Inputs/Value Channel 01 <-> Data Pointer/RawPositionValues[0]
//     Term 65 (AT2002-0250)/Term 66 (AT2002-5250)/FB Inputs/Value Channel 02 <-> Data Pointer/RawPositionValues[1]
//     Term 65 (AT2002-0250)/Term 66 (AT2002-5250)/FB Inputs/Value Channel 03 <-> Data Pointer/RawPositionValues[2]
//     Term 65 (AT2002-0250)/Term 66 (AT2002-5250)/FB Inputs/Value Channel 04 <-> Data Pointer/RawPositionValues[3]
//     Term 65 (AT2002-0250)/Term 66 (AT2002-5250)/FB Inputs/Value Channel 05 <-> Data Pointer/RawPositionValues[4]
//     Term 65 (AT2002-0250)/Term 66 (AT2002-5250)/FB Inputs/Value Channel 06 <-> Data Pointer/RawPositionValues[5]
//     Term 65 (AT2002-0250)/Term 66 (AT2002-5250)/FB Inputs/Value Channel 07 <-> Data Pointer/RawPositionValues[6]
//     Term 65 (AT2002-0250)/Term 66 (AT2002-5250)/FB Inputs/Value Channel 08 <-> Data Pointer/RawPositionValues[7]
//     Term 65 (AT2002-0250)/Term 66 (AT2002-5250)/FB Inputs/Value Channel 09 <-> Data Pointer/RawPositionValues[8]
//     Term 65 (AT2002-0250)/Term 66 (AT2002-5250)/FB Inputs/Value Channel 10 <-> Data Pointer/RawPositionValues[9]
//     Term 65 (AT2002-0250)/Term 66 (AT2002-5250)/FB Inputs/Value Channel 11 <-> Data Pointer/RawPositionValues[10]
//     Term 65 (AT2002-0250)/Term 66 (AT2002-5250)/FB Inputs/Value Channel 12 <-> Data Pointer/RawPositionValues[11]
//     Term 65 (AT2002-0250)/Term 66 (AT2002-5250)/FB Inputs/Value Channel 13 <-> Data Pointer/RawPositionValues[12]
//     Term 65 (AT2002-0250)/Term 66 (AT2002-5250)/FB Inputs/Value Channel 14 <-> Data Pointer/RawPositionValues[13]
//     Term 65 (AT2002-0250)/Term 66 (AT2002-5250)/FB Inputs/Value Channel 15 <-> Data Pointer/RawPositionValues[14]
//     Term 65 (AT2002-0250)/Term 66 (AT2002-5250)/FB Inputs/Value Channel 16 <-> Data Pointer/RawPositionValues[15]
//     Term 65 (AT2002-0250)/Term 66 (AT2002-5250)/FB Inputs/Value Channel 17 <-> Data Pointer/RawPositionValues[16]
//     Term 65 (AT2002-0250)/Term 66 (AT2002-5250)/FB Inputs/Value Channel 18 <-> Data Pointer/RawPositionValues[17]
//     Term 65 (AT2002-0250)/Term 66 (AT2002-5250)/FB Inputs/Value Channel 19 <-> Data Pointer/RawPositionValues[18]
//     Term 65 (AT2002-0250)/Term 66 (AT2002-5250)/FB Inputs/Value Channel 20 <-> Data Pointer/RawPositionValues[19]
//     Term 65 (AT2002-0250)/Term 66 (AT2002-5250)/FB Inputs/Value Channel 21 <-> Data Pointer/RawPositionValues[20]
//     Term 65 (AT2002-0250)/Term 66 (AT2002-5250)/FB Inputs/Value Channel 22 <-> Data Pointer/RawPositionValues[21]
//     Term 65 (AT2002-0250)/Term 66 (AT2002-5250)/FB Inputs/Value Channel 23 <-> Data Pointer/RawPositionValues[22]
//     Term 65 (AT2002-0250)/Term 66 (AT2002-5250)/FB Inputs/Value Channel 24 <-> Data Pointer/RawPositionValues[23]
//     Term 65 (AT2002-0250)/Term 66 (AT2002-5250)/FB Inputs/Value Channel 25 <-> Data Pointer/RawPositionValues[24]
//     Term 65 (AT2002-0250)/Term 66 (AT2002-5250)/FB Inputs/Value Channel 26 <-> Data Pointer/RawPositionValues[25]
//     Term 65 (AT2002-0250)/Term 66 (AT2002-5250)/FB Inputs/Value Channel 27 <-> Data Pointer/RawPositionValues[26]
//     Term 65 (AT2002-0250)/Term 66 (AT2002-5250)/FB Inputs/Value Channel 28 <-> Data Pointer/RawPositionValues[27]
//     Term 65 (AT2002-0250)/Term 66 (AT2002-5250)/FB Inputs/Value Channel 29 <-> Data Pointer/RawPositionValues[28]
//     Term 65 (AT2002-0250)/Term 66 (AT2002-5250)/FB Inputs/Value Channel 30 <-> Data Pointer/RawPositionValues[29]
//     Term 65 (AT2002-0250)/Term 66 (AT2002-5250)/FB Inputs/Value Channel 31 <-> Data Pointer/RawPositionValues[30]
//     Term 65 (AT2002-0250)/Term 66 (AT2002-5250)/FB Inputs/Value Channel 32 <-> Data Pointer/RawPositionValues[31]
//   Device 32 <-> TcCOM Objects/XTS ProcessingUnit 1/Part 1/Module 51
//     Term 67 (AT2200-0500)/CC Inputs/Current actual value Ch.1 <-> Data Pointer/CurrentActualValues[0]
//     Term 67 (AT2200-0500)/CC Inputs/Current actual value Ch.10 <-> Data Pointer/CurrentActualValues[9]
//     Term 67 (AT2200-0500)/CC Inputs/Current actual value Ch.11 <-> Data Pointer/CurrentActualValues[10]
//     Term 67 (AT2200-0500)/CC Inputs/Current actual value Ch.12 <-> Data Pointer/CurrentActualValues[11]
//     Term 67 (AT2200-0500)/CC Inputs/Current actual value Ch.13 <-> Data Pointer/CurrentActualValues[12]
//     Term 67 (AT2200-0500)/CC Inputs/Current actual value Ch.14 <-> Data Pointer/CurrentActualValues[13]
//     Term 67 (AT2200-0500)/CC Inputs/Current actual value Ch.15 <-> Data Pointer/CurrentActualValues[14]
//     Term 67 (AT2200-0500)/CC Inputs/Current actual value Ch.16 <-> Data Pointer/CurrentActualValues[15]
//     Term 67 (AT2200-0500)/CC Inputs/Current actual value Ch.17 <-> Data Pointer/CurrentActualValues[16]
//     Term 67 (AT2200-0500)/CC Inputs/Current actual value Ch.18 <-> Data Pointer/CurrentActualValues[17]
//     Term 67 (AT2200-0500)/CC Inputs/Current actual value Ch.19 <-> Data Pointer/CurrentActualValues[18]
//     Term 67 (AT2200-0500)/CC Inputs/Current actual value Ch.2 <-> Data Pointer/CurrentActualValues[1]
//     Term 67 (AT2200-0500)/CC Inputs/Current actual value Ch.20 <-> Data Pointer/CurrentActualValues[19]
//     Term 67 (AT2200-0500)/CC Inputs/Current actual value Ch.21 <-> Data Pointer/CurrentActualValues[20]
//     Term 67 (AT2200-0500)/CC Inputs/Current actual value Ch.22 <-> Data Pointer/CurrentActualValues[21]
//     Term 67 (AT2200-0500)/CC Inputs/Current actual value Ch.23 <-> Data Pointer/CurrentActualValues[22]
//     Term 67 (AT2200-0500)/CC Inputs/Current actual value Ch.24 <-> Data Pointer/CurrentActualValues[23]
//     Term 67 (AT2200-0500)/CC Inputs/Current actual value Ch.25 <-> Data Pointer/CurrentActualValues[24]
//     Term 67 (AT2200-0500)/CC Inputs/Current actual value Ch.26 <-> Data Pointer/CurrentActualValues[25]
//     Term 67 (AT2200-0500)/CC Inputs/Current actual value Ch.27 <-> Data Pointer/CurrentActualValues[26]
//     Term 67 (AT2200-0500)/CC Inputs/Current actual value Ch.28 <-> Data Pointer/CurrentActualValues[27]
//     Term 67 (AT2200-0500)/CC Inputs/Current actual value Ch.29 <-> Data Pointer/CurrentActualValues[28]
//     Term 67 (AT2200-0500)/CC Inputs/Current actual value Ch.3 <-> Data Pointer/CurrentActualValues[2]
//     Term 67 (AT2200-0500)/CC Inputs/Current actual value Ch.30 <-> Data Pointer/CurrentActualValues[29]
//     Term 67 (AT2200-0500)/CC Inputs/Current actual value Ch.4 <-> Data Pointer/CurrentActualValues[3]
//     Term 67 (AT2200-0500)/CC Inputs/Current actual value Ch.5 <-> Data Pointer/CurrentActualValues[4]
//     Term 67 (AT2200-0500)/CC Inputs/Current actual value Ch.6 <-> Data Pointer/CurrentActualValues[5]
//     Term 67 (AT2200-0500)/CC Inputs/Current actual value Ch.7 <-> Data Pointer/CurrentActualValues[6]
//     Term 67 (AT2200-0500)/CC Inputs/Current actual value Ch.8 <-> Data Pointer/CurrentActualValues[7]
//     Term 67 (AT2200-0500)/CC Inputs/Current actual value Ch.9 <-> Data Pointer/CurrentActualValues[8]
//     Term 67 (AT2200-0500)/CC Inputs/Status <-> Data Pointer/Status
//     Term 67 (AT2200-0500)/CC Outputs/Control <-> Data Pointer/Control
//     Term 67 (AT2200-0500)/CC Outputs/Current setpoint value Ch.1 <-> Data Pointer/CurrentSetpointValues[0]
//     Term 67 (AT2200-0500)/CC Outputs/Current setpoint value Ch.10 <-> Data Pointer/CurrentSetpointValues[9]
//     Term 67 (AT2200-0500)/CC Outputs/Current setpoint value Ch.11 <-> Data Pointer/CurrentSetpointValues[10]
//     Term 67 (AT2200-0500)/CC Outputs/Current setpoint value Ch.12 <-> Data Pointer/CurrentSetpointValues[11]
//     Term 67 (AT2200-0500)/CC Outputs/Current setpoint value Ch.13 <-> Data Pointer/CurrentSetpointValues[12]
//     Term 67 (AT2200-0500)/CC Outputs/Current setpoint value Ch.14 <-> Data Pointer/CurrentSetpointValues[13]
//     Term 67 (AT2200-0500)/CC Outputs/Current setpoint value Ch.15 <-> Data Pointer/CurrentSetpointValues[14]
//     Term 67 (AT2200-0500)/CC Outputs/Current setpoint value Ch.16 <-> Data Pointer/CurrentSetpointValues[15]
//     Term 67 (AT2200-0500)/CC Outputs/Current setpoint value Ch.17 <-> Data Pointer/CurrentSetpointValues[16]
//     Term 67 (AT2200-0500)/CC Outputs/Current setpoint value Ch.18 <-> Data Pointer/CurrentSetpointValues[17]
//     Term 67 (AT2200-0500)/CC Outputs/Current setpoint value Ch.19 <-> Data Pointer/CurrentSetpointValues[18]
//     Term 67 (AT2200-0500)/CC Outputs/Current setpoint value Ch.2 <-> Data Pointer/CurrentSetpointValues[1]
//     Term 67 (AT2200-0500)/CC Outputs/Current setpoint value Ch.20 <-> Data Pointer/CurrentSetpointValues[19]
//     Term 67 (AT2200-0500)/CC Outputs/Current setpoint value Ch.21 <-> Data Pointer/CurrentSetpointValues[20]
//     Term 67 (AT2200-0500)/CC Outputs/Current setpoint value Ch.22 <-> Data Pointer/CurrentSetpointValues[21]
//     Term 67 (AT2200-0500)/CC Outputs/Current setpoint value Ch.23 <-> Data Pointer/CurrentSetpointValues[22]
//     Term 67 (AT2200-0500)/CC Outputs/Current setpoint value Ch.24 <-> Data Pointer/CurrentSetpointValues[23]
//     Term 67 (AT2200-0500)/CC Outputs/Current setpoint value Ch.25 <-> Data Pointer/CurrentSetpointValues[24]
//     Term 67 (AT2200-0500)/CC Outputs/Current setpoint value Ch.26 <-> Data Pointer/CurrentSetpointValues[25]
//     Term 67 (AT2200-0500)/CC Outputs/Current setpoint value Ch.27 <-> Data Pointer/CurrentSetpointValues[26]
//     Term 67 (AT2200-0500)/CC Outputs/Current setpoint value Ch.28 <-> Data Pointer/CurrentSetpointValues[27]
//     Term 67 (AT2200-0500)/CC Outputs/Current setpoint value Ch.29 <-> Data Pointer/CurrentSetpointValues[28]
//     Term 67 (AT2200-0500)/CC Outputs/Current setpoint value Ch.3 <-> Data Pointer/CurrentSetpointValues[2]
//     Term 67 (AT2200-0500)/CC Outputs/Current setpoint value Ch.30 <-> Data Pointer/CurrentSetpointValues[29]
//     Term 67 (AT2200-0500)/CC Outputs/Current setpoint value Ch.4 <-> Data Pointer/CurrentSetpointValues[3]
//     Term 67 (AT2200-0500)/CC Outputs/Current setpoint value Ch.5 <-> Data Pointer/CurrentSetpointValues[4]
//     Term 67 (AT2200-0500)/CC Outputs/Current setpoint value Ch.6 <-> Data Pointer/CurrentSetpointValues[5]
//     Term 67 (AT2200-0500)/CC Outputs/Current setpoint value Ch.7 <-> Data Pointer/CurrentSetpointValues[6]
//     Term 67 (AT2200-0500)/CC Outputs/Current setpoint value Ch.8 <-> Data Pointer/CurrentSetpointValues[7]
//     Term 67 (AT2200-0500)/CC Outputs/Current setpoint value Ch.9 <-> Data Pointer/CurrentSetpointValues[8]
//     Term 67 (AT2200-0500)/LFB Inputs/BinaryData <-> Data Pointer/HallSensorValues
//   Device 32 <-> TcCOM Objects/XTS ProcessingUnit 1/Part 1/Module 52
//     Term 68 (AT2200-0500)/CC Inputs/Current actual value Ch.1 <-> Data Pointer/CurrentActualValues[0]
//     Term 68 (AT2200-0500)/CC Inputs/Current actual value Ch.10 <-> Data Pointer/CurrentActualValues[9]
//     Term 68 (AT2200-0500)/CC Inputs/Current actual value Ch.11 <-> Data Pointer/CurrentActualValues[10]
//     Term 68 (AT2200-0500)/CC Inputs/Current actual value Ch.12 <-> Data Pointer/CurrentActualValues[11]
//     Term 68 (AT2200-0500)/CC Inputs/Current actual value Ch.13 <-> Data Pointer/CurrentActualValues[12]
//     Term 68 (AT2200-0500)/CC Inputs/Current actual value Ch.14 <-> Data Pointer/CurrentActualValues[13]
//     Term 68 (AT2200-0500)/CC Inputs/Current actual value Ch.15 <-> Data Pointer/CurrentActualValues[14]
//     Term 68 (AT2200-0500)/CC Inputs/Current actual value Ch.16 <-> Data Pointer/CurrentActualValues[15]
//     Term 68 (AT2200-0500)/CC Inputs/Current actual value Ch.17 <-> Data Pointer/CurrentActualValues[16]
//     Term 68 (AT2200-0500)/CC Inputs/Current actual value Ch.18 <-> Data Pointer/CurrentActualValues[17]
//     Term 68 (AT2200-0500)/CC Inputs/Current actual value Ch.19 <-> Data Pointer/CurrentActualValues[18]
//     Term 68 (AT2200-0500)/CC Inputs/Current actual value Ch.2 <-> Data Pointer/CurrentActualValues[1]
//     Term 68 (AT2200-0500)/CC Inputs/Current actual value Ch.20 <-> Data Pointer/CurrentActualValues[19]
//     Term 68 (AT2200-0500)/CC Inputs/Current actual value Ch.21 <-> Data Pointer/CurrentActualValues[20]
//     Term 68 (AT2200-0500)/CC Inputs/Current actual value Ch.22 <-> Data Pointer/CurrentActualValues[21]
//     Term 68 (AT2200-0500)/CC Inputs/Current actual value Ch.23 <-> Data Pointer/CurrentActualValues[22]
//     Term 68 (AT2200-0500)/CC Inputs/Current actual value Ch.24 <-> Data Pointer/CurrentActualValues[23]
//     Term 68 (AT2200-0500)/CC Inputs/Current actual value Ch.25 <-> Data Pointer/CurrentActualValues[24]
//     Term 68 (AT2200-0500)/CC Inputs/Current actual value Ch.26 <-> Data Pointer/CurrentActualValues[25]
//     Term 68 (AT2200-0500)/CC Inputs/Current actual value Ch.27 <-> Data Pointer/CurrentActualValues[26]
//     Term 68 (AT2200-0500)/CC Inputs/Current actual value Ch.28 <-> Data Pointer/CurrentActualValues[27]
//     Term 68 (AT2200-0500)/CC Inputs/Current actual value Ch.29 <-> Data Pointer/CurrentActualValues[28]
//     Term 68 (AT2200-0500)/CC Inputs/Current actual value Ch.3 <-> Data Pointer/CurrentActualValues[2]
//     Term 68 (AT2200-0500)/CC Inputs/Current actual value Ch.30 <-> Data Pointer/CurrentActualValues[29]
//     Term 68 (AT2200-0500)/CC Inputs/Current actual value Ch.4 <-> Data Pointer/CurrentActualValues[3]
//     Term 68 (AT2200-0500)/CC Inputs/Current actual value Ch.5 <-> Data Pointer/CurrentActualValues[4]
//     Term 68 (AT2200-0500)/CC Inputs/Current actual value Ch.6 <-> Data Pointer/CurrentActualValues[5]
//     Term 68 (AT2200-0500)/CC Inputs/Current actual value Ch.7 <-> Data Pointer/CurrentActualValues[6]
//     Term 68 (AT2200-0500)/CC Inputs/Current actual value Ch.8 <-> Data Pointer/CurrentActualValues[7]
//     Term 68 (AT2200-0500)/CC Inputs/Current actual value Ch.9 <-> Data Pointer/CurrentActualValues[8]
//     Term 68 (AT2200-0500)/CC Inputs/Status <-> Data Pointer/Status
//     Term 68 (AT2200-0500)/CC Outputs/Control <-> Data Pointer/Control
//     Term 68 (AT2200-0500)/CC Outputs/Current setpoint value Ch.1 <-> Data Pointer/CurrentSetpointValues[0]
//     Term 68 (AT2200-0500)/CC Outputs/Current setpoint value Ch.10 <-> Data Pointer/CurrentSetpointValues[9]
//     Term 68 (AT2200-0500)/CC Outputs/Current setpoint value Ch.11 <-> Data Pointer/CurrentSetpointValues[10]
//     Term 68 (AT2200-0500)/CC Outputs/Current setpoint value Ch.12 <-> Data Pointer/CurrentSetpointValues[11]
//     Term 68 (AT2200-0500)/CC Outputs/Current setpoint value Ch.13 <-> Data Pointer/CurrentSetpointValues[12]
//     Term 68 (AT2200-0500)/CC Outputs/Current setpoint value Ch.14 <-> Data Pointer/CurrentSetpointValues[13]
//     Term 68 (AT2200-0500)/CC Outputs/Current setpoint value Ch.15 <-> Data Pointer/CurrentSetpointValues[14]
//     Term 68 (AT2200-0500)/CC Outputs/Current setpoint value Ch.16 <-> Data Pointer/CurrentSetpointValues[15]
//     Term 68 (AT2200-0500)/CC Outputs/Current setpoint value Ch.17 <-> Data Pointer/CurrentSetpointValues[16]
//     Term 68 (AT2200-0500)/CC Outputs/Current setpoint value Ch.18 <-> Data Pointer/CurrentSetpointValues[17]
//     Term 68 (AT2200-0500)/CC Outputs/Current setpoint value Ch.19 <-> Data Pointer/CurrentSetpointValues[18]
//     Term 68 (AT2200-0500)/CC Outputs/Current setpoint value Ch.2 <-> Data Pointer/CurrentSetpointValues[1]
//     Term 68 (AT2200-0500)/CC Outputs/Current setpoint value Ch.20 <-> Data Pointer/CurrentSetpointValues[19]
//     Term 68 (AT2200-0500)/CC Outputs/Current setpoint value Ch.21 <-> Data Pointer/CurrentSetpointValues[20]
//     Term 68 (AT2200-0500)/CC Outputs/Current setpoint value Ch.22 <-> Data Pointer/CurrentSetpointValues[21]
//     Term 68 (AT2200-0500)/CC Outputs/Current setpoint value Ch.23 <-> Data Pointer/CurrentSetpointValues[22]
//     Term 68 (AT2200-0500)/CC Outputs/Current setpoint value Ch.24 <-> Data Pointer/CurrentSetpointValues[23]
//     Term 68 (AT2200-0500)/CC Outputs/Current setpoint value Ch.25 <-> Data Pointer/CurrentSetpointValues[24]
//     Term 68 (AT2200-0500)/CC Outputs/Current setpoint value Ch.26 <-> Data Pointer/CurrentSetpointValues[25]
//     Term 68 (AT2200-0500)/CC Outputs/Current setpoint value Ch.27 <-> Data Pointer/CurrentSetpointValues[26]
//     Term 68 (AT2200-0500)/CC Outputs/Current setpoint value Ch.28 <-> Data Pointer/CurrentSetpointValues[27]
//     Term 68 (AT2200-0500)/CC Outputs/Current setpoint value Ch.29 <-> Data Pointer/CurrentSetpointValues[28]
//     Term 68 (AT2200-0500)/CC Outputs/Current setpoint value Ch.3 <-> Data Pointer/CurrentSetpointValues[2]
//     Term 68 (AT2200-0500)/CC Outputs/Current setpoint value Ch.30 <-> Data Pointer/CurrentSetpointValues[29]
//     Term 68 (AT2200-0500)/CC Outputs/Current setpoint value Ch.4 <-> Data Pointer/CurrentSetpointValues[3]
//     Term 68 (AT2200-0500)/CC Outputs/Current setpoint value Ch.5 <-> Data Pointer/CurrentSetpointValues[4]
//     Term 68 (AT2200-0500)/CC Outputs/Current setpoint value Ch.6 <-> Data Pointer/CurrentSetpointValues[5]
//     Term 68 (AT2200-0500)/CC Outputs/Current setpoint value Ch.7 <-> Data Pointer/CurrentSetpointValues[6]
//     Term 68 (AT2200-0500)/CC Outputs/Current setpoint value Ch.8 <-> Data Pointer/CurrentSetpointValues[7]
//     Term 68 (AT2200-0500)/CC Outputs/Current setpoint value Ch.9 <-> Data Pointer/CurrentSetpointValues[8]
//     Term 68 (AT2200-0500)/LFB Inputs/BinaryData <-> Data Pointer/HallSensorValues
//   Device 33 <-> TcCOM Objects/XTS ProcessingUnit 1/Part 1/Module 53
//     Term 69 (AT2042-0250)/CC Inputs/Current actual value Ch.1 <-> Data Pointer/CurrentActualValues[0]
//     Term 69 (AT2042-0250)/CC Inputs/Current actual value Ch.10 <-> Data Pointer/CurrentActualValues[9]
//     Term 69 (AT2042-0250)/CC Inputs/Current actual value Ch.11 <-> Data Pointer/CurrentActualValues[10]
//     Term 69 (AT2042-0250)/CC Inputs/Current actual value Ch.12 <-> Data Pointer/CurrentActualValues[11]
//     Term 69 (AT2042-0250)/CC Inputs/Current actual value Ch.13 <-> Data Pointer/CurrentActualValues[12]
//     Term 69 (AT2042-0250)/CC Inputs/Current actual value Ch.14 <-> Data Pointer/CurrentActualValues[13]
//     Term 69 (AT2042-0250)/CC Inputs/Current actual value Ch.15 <-> Data Pointer/CurrentActualValues[14]
//     Term 69 (AT2042-0250)/CC Inputs/Current actual value Ch.2 <-> Data Pointer/CurrentActualValues[1]
//     Term 69 (AT2042-0250)/CC Inputs/Current actual value Ch.3 <-> Data Pointer/CurrentActualValues[2]
//     Term 69 (AT2042-0250)/CC Inputs/Current actual value Ch.4 <-> Data Pointer/CurrentActualValues[3]
//     Term 69 (AT2042-0250)/CC Inputs/Current actual value Ch.5 <-> Data Pointer/CurrentActualValues[4]
//     Term 69 (AT2042-0250)/CC Inputs/Current actual value Ch.6 <-> Data Pointer/CurrentActualValues[5]
//     Term 69 (AT2042-0250)/CC Inputs/Current actual value Ch.7 <-> Data Pointer/CurrentActualValues[6]
//     Term 69 (AT2042-0250)/CC Inputs/Current actual value Ch.8 <-> Data Pointer/CurrentActualValues[7]
//     Term 69 (AT2042-0250)/CC Inputs/Current actual value Ch.9 <-> Data Pointer/CurrentActualValues[8]
//     Term 69 (AT2042-0250)/CC Inputs/Status <-> Data Pointer/Status
//     Term 69 (AT2042-0250)/CC Outputs/Control <-> Data Pointer/Control
//     Term 69 (AT2042-0250)/CC Outputs/Current setpoint value Ch.1 <-> Data Pointer/CurrentSetpointValues[0]
//     Term 69 (AT2042-0250)/CC Outputs/Current setpoint value Ch.10 <-> Data Pointer/CurrentSetpointValues[9]
//     Term 69 (AT2042-0250)/CC Outputs/Current setpoint value Ch.11 <-> Data Pointer/CurrentSetpointValues[10]
//     Term 69 (AT2042-0250)/CC Outputs/Current setpoint value Ch.12 <-> Data Pointer/CurrentSetpointValues[11]
//     Term 69 (AT2042-0250)/CC Outputs/Current setpoint value Ch.13 <-> Data Pointer/CurrentSetpointValues[12]
//     Term 69 (AT2042-0250)/CC Outputs/Current setpoint value Ch.14 <-> Data Pointer/CurrentSetpointValues[13]
//     Term 69 (AT2042-0250)/CC Outputs/Current setpoint value Ch.15 <-> Data Pointer/CurrentSetpointValues[14]
//     Term 69 (AT2042-0250)/CC Outputs/Current setpoint value Ch.2 <-> Data Pointer/CurrentSetpointValues[1]
//     Term 69 (AT2042-0250)/CC Outputs/Current setpoint value Ch.3 <-> Data Pointer/CurrentSetpointValues[2]
//     Term 69 (AT2042-0250)/CC Outputs/Current setpoint value Ch.4 <-> Data Pointer/CurrentSetpointValues[3]
//     Term 69 (AT2042-0250)/CC Outputs/Current setpoint value Ch.5 <-> Data Pointer/CurrentSetpointValues[4]
//     Term 69 (AT2042-0250)/CC Outputs/Current setpoint value Ch.6 <-> Data Pointer/CurrentSetpointValues[5]
//     Term 69 (AT2042-0250)/CC Outputs/Current setpoint value Ch.7 <-> Data Pointer/CurrentSetpointValues[6]
//     Term 69 (AT2042-0250)/CC Outputs/Current setpoint value Ch.8 <-> Data Pointer/CurrentSetpointValues[7]
//     Term 69 (AT2042-0250)/CC Outputs/Current setpoint value Ch.9 <-> Data Pointer/CurrentSetpointValues[8]
//     Term 69 (AT2042-0250)/Term 70 (AT2042-5250)/FB Inputs/Value Channel 01 <-> Data Pointer/RawPositionValues[0]
//     Term 69 (AT2042-0250)/Term 70 (AT2042-5250)/FB Inputs/Value Channel 02 <-> Data Pointer/RawPositionValues[1]
//     Term 69 (AT2042-0250)/Term 70 (AT2042-5250)/FB Inputs/Value Channel 03 <-> Data Pointer/RawPositionValues[2]
//     Term 69 (AT2042-0250)/Term 70 (AT2042-5250)/FB Inputs/Value Channel 04 <-> Data Pointer/RawPositionValues[3]
//     Term 69 (AT2042-0250)/Term 70 (AT2042-5250)/FB Inputs/Value Channel 05 <-> Data Pointer/RawPositionValues[4]
//     Term 69 (AT2042-0250)/Term 70 (AT2042-5250)/FB Inputs/Value Channel 06 <-> Data Pointer/RawPositionValues[5]
//     Term 69 (AT2042-0250)/Term 70 (AT2042-5250)/FB Inputs/Value Channel 07 <-> Data Pointer/RawPositionValues[6]
//     Term 69 (AT2042-0250)/Term 70 (AT2042-5250)/FB Inputs/Value Channel 08 <-> Data Pointer/RawPositionValues[7]
//     Term 69 (AT2042-0250)/Term 70 (AT2042-5250)/FB Inputs/Value Channel 09 <-> Data Pointer/RawPositionValues[8]
//     Term 69 (AT2042-0250)/Term 70 (AT2042-5250)/FB Inputs/Value Channel 10 <-> Data Pointer/RawPositionValues[9]
//     Term 69 (AT2042-0250)/Term 70 (AT2042-5250)/FB Inputs/Value Channel 11 <-> Data Pointer/RawPositionValues[10]
//     Term 69 (AT2042-0250)/Term 70 (AT2042-5250)/FB Inputs/Value Channel 12 <-> Data Pointer/RawPositionValues[11]
//     Term 69 (AT2042-0250)/Term 70 (AT2042-5250)/FB Inputs/Value Channel 13 <-> Data Pointer/RawPositionValues[12]
//     Term 69 (AT2042-0250)/Term 70 (AT2042-5250)/FB Inputs/Value Channel 14 <-> Data Pointer/RawPositionValues[13]
//     Term 69 (AT2042-0250)/Term 70 (AT2042-5250)/FB Inputs/Value Channel 15 <-> Data Pointer/RawPositionValues[14]
//     Term 69 (AT2042-0250)/Term 70 (AT2042-5250)/FB Inputs/Value Channel 16 <-> Data Pointer/RawPositionValues[15]
//     Term 69 (AT2042-0250)/Term 70 (AT2042-5250)/FB Inputs/Value Channel 17 <-> Data Pointer/RawPositionValues[16]
//     Term 69 (AT2042-0250)/Term 70 (AT2042-5250)/FB Inputs/Value Channel 18 <-> Data Pointer/RawPositionValues[17]
//     Term 69 (AT2042-0250)/Term 70 (AT2042-5250)/FB Inputs/Value Channel 19 <-> Data Pointer/RawPositionValues[18]
//     Term 69 (AT2042-0250)/Term 70 (AT2042-5250)/FB Inputs/Value Channel 20 <-> Data Pointer/RawPositionValues[19]
//     Term 69 (AT2042-0250)/Term 70 (AT2042-5250)/FB Inputs/Value Channel 21 <-> Data Pointer/RawPositionValues[20]
//     Term 69 (AT2042-0250)/Term 70 (AT2042-5250)/FB Inputs/Value Channel 22 <-> Data Pointer/RawPositionValues[21]
//     Term 69 (AT2042-0250)/Term 70 (AT2042-5250)/FB Inputs/Value Channel 23 <-> Data Pointer/RawPositionValues[22]
//     Term 69 (AT2042-0250)/Term 70 (AT2042-5250)/FB Inputs/Value Channel 24 <-> Data Pointer/RawPositionValues[23]
//     Term 69 (AT2042-0250)/Term 70 (AT2042-5250)/FB Inputs/Value Channel 25 <-> Data Pointer/RawPositionValues[24]
//     Term 69 (AT2042-0250)/Term 70 (AT2042-5250)/FB Inputs/Value Channel 26 <-> Data Pointer/RawPositionValues[25]
//     Term 69 (AT2042-0250)/Term 70 (AT2042-5250)/FB Inputs/Value Channel 27 <-> Data Pointer/RawPositionValues[26]
//     Term 69 (AT2042-0250)/Term 70 (AT2042-5250)/FB Inputs/Value Channel 28 <-> Data Pointer/RawPositionValues[27]
//     Term 69 (AT2042-0250)/Term 70 (AT2042-5250)/FB Inputs/Value Channel 29 <-> Data Pointer/RawPositionValues[28]
//     Term 69 (AT2042-0250)/Term 70 (AT2042-5250)/FB Inputs/Value Channel 30 <-> Data Pointer/RawPositionValues[29]
//     Term 69 (AT2042-0250)/Term 70 (AT2042-5250)/FB Inputs/Value Channel 31 <-> Data Pointer/RawPositionValues[30]
//     Term 69 (AT2042-0250)/Term 70 (AT2042-5250)/FB Inputs/Value Channel 32 <-> Data Pointer/RawPositionValues[31]
//   Device 33 <-> TcCOM Objects/XTS ProcessingUnit 1/Part 1/Module 54
//     Term 71 (AT2040-0250)/CC Inputs/Current actual value Ch.1 <-> Data Pointer/CurrentActualValues[0]
//     Term 71 (AT2040-0250)/CC Inputs/Current actual value Ch.10 <-> Data Pointer/CurrentActualValues[9]
//     Term 71 (AT2040-0250)/CC Inputs/Current actual value Ch.11 <-> Data Pointer/CurrentActualValues[10]
//     Term 71 (AT2040-0250)/CC Inputs/Current actual value Ch.12 <-> Data Pointer/CurrentActualValues[11]
//     Term 71 (AT2040-0250)/CC Inputs/Current actual value Ch.13 <-> Data Pointer/CurrentActualValues[12]
//     Term 71 (AT2040-0250)/CC Inputs/Current actual value Ch.14 <-> Data Pointer/CurrentActualValues[13]
//     Term 71 (AT2040-0250)/CC Inputs/Current actual value Ch.15 <-> Data Pointer/CurrentActualValues[14]
//     Term 71 (AT2040-0250)/CC Inputs/Current actual value Ch.2 <-> Data Pointer/CurrentActualValues[1]
//     Term 71 (AT2040-0250)/CC Inputs/Current actual value Ch.3 <-> Data Pointer/CurrentActualValues[2]
//     Term 71 (AT2040-0250)/CC Inputs/Current actual value Ch.4 <-> Data Pointer/CurrentActualValues[3]
//     Term 71 (AT2040-0250)/CC Inputs/Current actual value Ch.5 <-> Data Pointer/CurrentActualValues[4]
//     Term 71 (AT2040-0250)/CC Inputs/Current actual value Ch.6 <-> Data Pointer/CurrentActualValues[5]
//     Term 71 (AT2040-0250)/CC Inputs/Current actual value Ch.7 <-> Data Pointer/CurrentActualValues[6]
//     Term 71 (AT2040-0250)/CC Inputs/Current actual value Ch.8 <-> Data Pointer/CurrentActualValues[7]
//     Term 71 (AT2040-0250)/CC Inputs/Current actual value Ch.9 <-> Data Pointer/CurrentActualValues[8]
//     Term 71 (AT2040-0250)/CC Inputs/Status <-> Data Pointer/Status
//     Term 71 (AT2040-0250)/CC Outputs/Control <-> Data Pointer/Control
//     Term 71 (AT2040-0250)/CC Outputs/Current setpoint value Ch.1 <-> Data Pointer/CurrentSetpointValues[0]
//     Term 71 (AT2040-0250)/CC Outputs/Current setpoint value Ch.10 <-> Data Pointer/CurrentSetpointValues[9]
//     Term 71 (AT2040-0250)/CC Outputs/Current setpoint value Ch.11 <-> Data Pointer/CurrentSetpointValues[10]
//     Term 71 (AT2040-0250)/CC Outputs/Current setpoint value Ch.12 <-> Data Pointer/CurrentSetpointValues[11]
//     Term 71 (AT2040-0250)/CC Outputs/Current setpoint value Ch.13 <-> Data Pointer/CurrentSetpointValues[12]
//     Term 71 (AT2040-0250)/CC Outputs/Current setpoint value Ch.14 <-> Data Pointer/CurrentSetpointValues[13]
//     Term 71 (AT2040-0250)/CC Outputs/Current setpoint value Ch.15 <-> Data Pointer/CurrentSetpointValues[14]
//     Term 71 (AT2040-0250)/CC Outputs/Current setpoint value Ch.2 <-> Data Pointer/CurrentSetpointValues[1]
//     Term 71 (AT2040-0250)/CC Outputs/Current setpoint value Ch.3 <-> Data Pointer/CurrentSetpointValues[2]
//     Term 71 (AT2040-0250)/CC Outputs/Current setpoint value Ch.4 <-> Data Pointer/CurrentSetpointValues[3]
//     Term 71 (AT2040-0250)/CC Outputs/Current setpoint value Ch.5 <-> Data Pointer/CurrentSetpointValues[4]
//     Term 71 (AT2040-0250)/CC Outputs/Current setpoint value Ch.6 <-> Data Pointer/CurrentSetpointValues[5]
//     Term 71 (AT2040-0250)/CC Outputs/Current setpoint value Ch.7 <-> Data Pointer/CurrentSetpointValues[6]
//     Term 71 (AT2040-0250)/CC Outputs/Current setpoint value Ch.8 <-> Data Pointer/CurrentSetpointValues[7]
//     Term 71 (AT2040-0250)/CC Outputs/Current setpoint value Ch.9 <-> Data Pointer/CurrentSetpointValues[8]
//     Term 71 (AT2040-0250)/Term 72 (AT2040-5250)/FB Inputs/Value Channel 01 <-> Data Pointer/RawPositionValues[0]
//     Term 71 (AT2040-0250)/Term 72 (AT2040-5250)/FB Inputs/Value Channel 02 <-> Data Pointer/RawPositionValues[1]
//     Term 71 (AT2040-0250)/Term 72 (AT2040-5250)/FB Inputs/Value Channel 03 <-> Data Pointer/RawPositionValues[2]
//     Term 71 (AT2040-0250)/Term 72 (AT2040-5250)/FB Inputs/Value Channel 04 <-> Data Pointer/RawPositionValues[3]
//     Term 71 (AT2040-0250)/Term 72 (AT2040-5250)/FB Inputs/Value Channel 05 <-> Data Pointer/RawPositionValues[4]
//     Term 71 (AT2040-0250)/Term 72 (AT2040-5250)/FB Inputs/Value Channel 06 <-> Data Pointer/RawPositionValues[5]
//     Term 71 (AT2040-0250)/Term 72 (AT2040-5250)/FB Inputs/Value Channel 07 <-> Data Pointer/RawPositionValues[6]
//     Term 71 (AT2040-0250)/Term 72 (AT2040-5250)/FB Inputs/Value Channel 08 <-> Data Pointer/RawPositionValues[7]
//     Term 71 (AT2040-0250)/Term 72 (AT2040-5250)/FB Inputs/Value Channel 09 <-> Data Pointer/RawPositionValues[8]
//     Term 71 (AT2040-0250)/Term 72 (AT2040-5250)/FB Inputs/Value Channel 10 <-> Data Pointer/RawPositionValues[9]
//     Term 71 (AT2040-0250)/Term 72 (AT2040-5250)/FB Inputs/Value Channel 11 <-> Data Pointer/RawPositionValues[10]
//     Term 71 (AT2040-0250)/Term 72 (AT2040-5250)/FB Inputs/Value Channel 12 <-> Data Pointer/RawPositionValues[11]
//     Term 71 (AT2040-0250)/Term 72 (AT2040-5250)/FB Inputs/Value Channel 13 <-> Data Pointer/RawPositionValues[12]
//     Term 71 (AT2040-0250)/Term 72 (AT2040-5250)/FB Inputs/Value Channel 14 <-> Data Pointer/RawPositionValues[13]
//     Term 71 (AT2040-0250)/Term 72 (AT2040-5250)/FB Inputs/Value Channel 15 <-> Data Pointer/RawPositionValues[14]
//     Term 71 (AT2040-0250)/Term 72 (AT2040-5250)/FB Inputs/Value Channel 16 <-> Data Pointer/RawPositionValues[15]
//     Term 71 (AT2040-0250)/Term 72 (AT2040-5250)/FB Inputs/Value Channel 17 <-> Data Pointer/RawPositionValues[16]
//     Term 71 (AT2040-0250)/Term 72 (AT2040-5250)/FB Inputs/Value Channel 18 <-> Data Pointer/RawPositionValues[17]
//     Term 71 (AT2040-0250)/Term 72 (AT2040-5250)/FB Inputs/Value Channel 19 <-> Data Pointer/RawPositionValues[18]
//     Term 71 (AT2040-0250)/Term 72 (AT2040-5250)/FB Inputs/Value Channel 20 <-> Data Pointer/RawPositionValues[19]
//     Term 71 (AT2040-0250)/Term 72 (AT2040-5250)/FB Inputs/Value Channel 21 <-> Data Pointer/RawPositionValues[20]
//     Term 71 (AT2040-0250)/Term 72 (AT2040-5250)/FB Inputs/Value Channel 22 <-> Data Pointer/RawPositionValues[21]
//     Term 71 (AT2040-0250)/Term 72 (AT2040-5250)/FB Inputs/Value Channel 23 <-> Data Pointer/RawPositionValues[22]
//     Term 71 (AT2040-0250)/Term 72 (AT2040-5250)/FB Inputs/Value Channel 24 <-> Data Pointer/RawPositionValues[23]
//     Term 71 (AT2040-0250)/Term 72 (AT2040-5250)/FB Inputs/Value Channel 25 <-> Data Pointer/RawPositionValues[24]
//     Term 71 (AT2040-0250)/Term 72 (AT2040-5250)/FB Inputs/Value Channel 26 <-> Data Pointer/RawPositionValues[25]
//     Term 71 (AT2040-0250)/Term 72 (AT2040-5250)/FB Inputs/Value Channel 27 <-> Data Pointer/RawPositionValues[26]
//     Term 71 (AT2040-0250)/Term 72 (AT2040-5250)/FB Inputs/Value Channel 28 <-> Data Pointer/RawPositionValues[27]
//     Term 71 (AT2040-0250)/Term 72 (AT2040-5250)/FB Inputs/Value Channel 29 <-> Data Pointer/RawPositionValues[28]
//     Term 71 (AT2040-0250)/Term 72 (AT2040-5250)/FB Inputs/Value Channel 30 <-> Data Pointer/RawPositionValues[29]
//     Term 71 (AT2040-0250)/Term 72 (AT2040-5250)/FB Inputs/Value Channel 31 <-> Data Pointer/RawPositionValues[30]
//     Term 71 (AT2040-0250)/Term 72 (AT2040-5250)/FB Inputs/Value Channel 32 <-> Data Pointer/RawPositionValues[31]
//   Device 33 <-> TcCOM Objects/XTS ProcessingUnit 1/Part 1/Module 55
//     Term 73 (AT2200-0500)/CC Inputs/Current actual value Ch.1 <-> Data Pointer/CurrentActualValues[0]
//     Term 73 (AT2200-0500)/CC Inputs/Current actual value Ch.10 <-> Data Pointer/CurrentActualValues[9]
//     Term 73 (AT2200-0500)/CC Inputs/Current actual value Ch.11 <-> Data Pointer/CurrentActualValues[10]
//     Term 73 (AT2200-0500)/CC Inputs/Current actual value Ch.12 <-> Data Pointer/CurrentActualValues[11]
//     Term 73 (AT2200-0500)/CC Inputs/Current actual value Ch.13 <-> Data Pointer/CurrentActualValues[12]
//     Term 73 (AT2200-0500)/CC Inputs/Current actual value Ch.14 <-> Data Pointer/CurrentActualValues[13]
//     Term 73 (AT2200-0500)/CC Inputs/Current actual value Ch.15 <-> Data Pointer/CurrentActualValues[14]
//     Term 73 (AT2200-0500)/CC Inputs/Current actual value Ch.16 <-> Data Pointer/CurrentActualValues[15]
//     Term 73 (AT2200-0500)/CC Inputs/Current actual value Ch.17 <-> Data Pointer/CurrentActualValues[16]
//     Term 73 (AT2200-0500)/CC Inputs/Current actual value Ch.18 <-> Data Pointer/CurrentActualValues[17]
//     Term 73 (AT2200-0500)/CC Inputs/Current actual value Ch.19 <-> Data Pointer/CurrentActualValues[18]
//     Term 73 (AT2200-0500)/CC Inputs/Current actual value Ch.2 <-> Data Pointer/CurrentActualValues[1]
//     Term 73 (AT2200-0500)/CC Inputs/Current actual value Ch.20 <-> Data Pointer/CurrentActualValues[19]
//     Term 73 (AT2200-0500)/CC Inputs/Current actual value Ch.21 <-> Data Pointer/CurrentActualValues[20]
//     Term 73 (AT2200-0500)/CC Inputs/Current actual value Ch.22 <-> Data Pointer/CurrentActualValues[21]
//     Term 73 (AT2200-0500)/CC Inputs/Current actual value Ch.23 <-> Data Pointer/CurrentActualValues[22]
//     Term 73 (AT2200-0500)/CC Inputs/Current actual value Ch.24 <-> Data Pointer/CurrentActualValues[23]
//     Term 73 (AT2200-0500)/CC Inputs/Current actual value Ch.25 <-> Data Pointer/CurrentActualValues[24]
//     Term 73 (AT2200-0500)/CC Inputs/Current actual value Ch.26 <-> Data Pointer/CurrentActualValues[25]
//     Term 73 (AT2200-0500)/CC Inputs/Current actual value Ch.27 <-> Data Pointer/CurrentActualValues[26]
//     Term 73 (AT2200-0500)/CC Inputs/Current actual value Ch.28 <-> Data Pointer/CurrentActualValues[27]
//     Term 73 (AT2200-0500)/CC Inputs/Current actual value Ch.29 <-> Data Pointer/CurrentActualValues[28]
//     Term 73 (AT2200-0500)/CC Inputs/Current actual value Ch.3 <-> Data Pointer/CurrentActualValues[2]
//     Term 73 (AT2200-0500)/CC Inputs/Current actual value Ch.30 <-> Data Pointer/CurrentActualValues[29]
//     Term 73 (AT2200-0500)/CC Inputs/Current actual value Ch.4 <-> Data Pointer/CurrentActualValues[3]
//     Term 73 (AT2200-0500)/CC Inputs/Current actual value Ch.5 <-> Data Pointer/CurrentActualValues[4]
//     Term 73 (AT2200-0500)/CC Inputs/Current actual value Ch.6 <-> Data Pointer/CurrentActualValues[5]
//     Term 73 (AT2200-0500)/CC Inputs/Current actual value Ch.7 <-> Data Pointer/CurrentActualValues[6]
//     Term 73 (AT2200-0500)/CC Inputs/Current actual value Ch.8 <-> Data Pointer/CurrentActualValues[7]
//     Term 73 (AT2200-0500)/CC Inputs/Current actual value Ch.9 <-> Data Pointer/CurrentActualValues[8]
//     Term 73 (AT2200-0500)/CC Inputs/Status <-> Data Pointer/Status
//     Term 73 (AT2200-0500)/CC Outputs/Control <-> Data Pointer/Control
//     Term 73 (AT2200-0500)/CC Outputs/Current setpoint value Ch.1 <-> Data Pointer/CurrentSetpointValues[0]
//     Term 73 (AT2200-0500)/CC Outputs/Current setpoint value Ch.10 <-> Data Pointer/CurrentSetpointValues[9]
//     Term 73 (AT2200-0500)/CC Outputs/Current setpoint value Ch.11 <-> Data Pointer/CurrentSetpointValues[10]
//     Term 73 (AT2200-0500)/CC Outputs/Current setpoint value Ch.12 <-> Data Pointer/CurrentSetpointValues[11]
//     Term 73 (AT2200-0500)/CC Outputs/Current setpoint value Ch.13 <-> Data Pointer/CurrentSetpointValues[12]
//     Term 73 (AT2200-0500)/CC Outputs/Current setpoint value Ch.14 <-> Data Pointer/CurrentSetpointValues[13]
//     Term 73 (AT2200-0500)/CC Outputs/Current setpoint value Ch.15 <-> Data Pointer/CurrentSetpointValues[14]
//     Term 73 (AT2200-0500)/CC Outputs/Current setpoint value Ch.16 <-> Data Pointer/CurrentSetpointValues[15]
//     Term 73 (AT2200-0500)/CC Outputs/Current setpoint value Ch.17 <-> Data Pointer/CurrentSetpointValues[16]
//     Term 73 (AT2200-0500)/CC Outputs/Current setpoint value Ch.18 <-> Data Pointer/CurrentSetpointValues[17]
//     Term 73 (AT2200-0500)/CC Outputs/Current setpoint value Ch.19 <-> Data Pointer/CurrentSetpointValues[18]
//     Term 73 (AT2200-0500)/CC Outputs/Current setpoint value Ch.2 <-> Data Pointer/CurrentSetpointValues[1]
//     Term 73 (AT2200-0500)/CC Outputs/Current setpoint value Ch.20 <-> Data Pointer/CurrentSetpointValues[19]
//     Term 73 (AT2200-0500)/CC Outputs/Current setpoint value Ch.21 <-> Data Pointer/CurrentSetpointValues[20]
//     Term 73 (AT2200-0500)/CC Outputs/Current setpoint value Ch.22 <-> Data Pointer/CurrentSetpointValues[21]
//     Term 73 (AT2200-0500)/CC Outputs/Current setpoint value Ch.23 <-> Data Pointer/CurrentSetpointValues[22]
//     Term 73 (AT2200-0500)/CC Outputs/Current setpoint value Ch.24 <-> Data Pointer/CurrentSetpointValues[23]
//     Term 73 (AT2200-0500)/CC Outputs/Current setpoint value Ch.25 <-> Data Pointer/CurrentSetpointValues[24]
//     Term 73 (AT2200-0500)/CC Outputs/Current setpoint value Ch.26 <-> Data Pointer/CurrentSetpointValues[25]
//     Term 73 (AT2200-0500)/CC Outputs/Current setpoint value Ch.27 <-> Data Pointer/CurrentSetpointValues[26]
//     Term 73 (AT2200-0500)/CC Outputs/Current setpoint value Ch.28 <-> Data Pointer/CurrentSetpointValues[27]
//     Term 73 (AT2200-0500)/CC Outputs/Current setpoint value Ch.29 <-> Data Pointer/CurrentSetpointValues[28]
//     Term 73 (AT2200-0500)/CC Outputs/Current setpoint value Ch.3 <-> Data Pointer/CurrentSetpointValues[2]
//     Term 73 (AT2200-0500)/CC Outputs/Current setpoint value Ch.30 <-> Data Pointer/CurrentSetpointValues[29]
//     Term 73 (AT2200-0500)/CC Outputs/Current setpoint value Ch.4 <-> Data Pointer/CurrentSetpointValues[3]
//     Term 73 (AT2200-0500)/CC Outputs/Current setpoint value Ch.5 <-> Data Pointer/CurrentSetpointValues[4]
//     Term 73 (AT2200-0500)/CC Outputs/Current setpoint value Ch.6 <-> Data Pointer/CurrentSetpointValues[5]
//     Term 73 (AT2200-0500)/CC Outputs/Current setpoint value Ch.7 <-> Data Pointer/CurrentSetpointValues[6]
//     Term 73 (AT2200-0500)/CC Outputs/Current setpoint value Ch.8 <-> Data Pointer/CurrentSetpointValues[7]
//     Term 73 (AT2200-0500)/CC Outputs/Current setpoint value Ch.9 <-> Data Pointer/CurrentSetpointValues[8]
//     Term 73 (AT2200-0500)/LFB Inputs/BinaryData <-> Data Pointer/HallSensorValues
//   ExternControl/ExternControl Instance <-> XtsTransport/XtsTransport Instance
//     PlcTask Inputs/MAIN_APP.eInitXtsTransport <-> PlcTask Outputs/MAIN_APP.eInit
//     PlcTask Inputs/MAPPING_in.StationState.byState <-> PlcTask Outputs/MAPPING_XTS_out.StationState.byState
//     PlcTask Inputs/MAPPING_in.TransportState.byState <-> PlcTask Outputs/MAPPING_XTS_out.TransportState.byState
//     PlcTask Outputs/MAPPING_out.StationControl.byCtrl <-> PlcTask Inputs/MAPPING_XTS_in.StationControl.byCtrl
//     PlcTask Outputs/MAPPING_out.TransportControl.byCtrl <-> PlcTask Inputs/MAPPING_XTS_in.TransportControl.byCtrl
//   XtsTransport/XtsTransport Instance <-> NC-Task 1/Axes/Mover Axis 1
//     PlcTask Inputs/GVL_XTS.AxisRefMover[1].NcToPlc <-> Outputs/ToPlc
//     PlcTask Outputs/GVL_XTS.AxisRefMover[1].PlcToNc <-> Inputs/FromPlc
//   XtsTransport/XtsTransport Instance <-> NC-Task 1/Axes/Mover Axis 10
//     PlcTask Inputs/GVL_XTS.AxisRefMover[10].NcToPlc <-> Outputs/ToPlc
//     PlcTask Outputs/GVL_XTS.AxisRefMover[10].PlcToNc <-> Inputs/FromPlc
//   XtsTransport/XtsTransport Instance <-> NC-Task 1/Axes/Mover Axis 100
//     PlcTask Inputs/GVL_XTS.AxisRefMover[100].NcToPlc <-> Outputs/ToPlc
//     PlcTask Outputs/GVL_XTS.AxisRefMover[100].PlcToNc <-> Inputs/FromPlc
//   XtsTransport/XtsTransport Instance <-> NC-Task 1/Axes/Mover Axis 101
//     PlcTask Inputs/GVL_XTS.AxisRefMover[101].NcToPlc <-> Outputs/ToPlc
//     PlcTask Outputs/GVL_XTS.AxisRefMover[101].PlcToNc <-> Inputs/FromPlc
//   XtsTransport/XtsTransport Instance <-> NC-Task 1/Axes/Mover Axis 102
//     PlcTask Inputs/GVL_XTS.AxisRefMover[102].NcToPlc <-> Outputs/ToPlc
//     PlcTask Outputs/GVL_XTS.AxisRefMover[102].PlcToNc <-> Inputs/FromPlc
//   XtsTransport/XtsTransport Instance <-> NC-Task 1/Axes/Mover Axis 103
//     PlcTask Inputs/GVL_XTS.AxisRefMover[103].NcToPlc <-> Outputs/ToPlc
//     PlcTask Outputs/GVL_XTS.AxisRefMover[103].PlcToNc <-> Inputs/FromPlc
//   XtsTransport/XtsTransport Instance <-> NC-Task 1/Axes/Mover Axis 104
//     PlcTask Inputs/GVL_XTS.AxisRefMover[104].NcToPlc <-> Outputs/ToPlc
//     PlcTask Outputs/GVL_XTS.AxisRefMover[104].PlcToNc <-> Inputs/FromPlc
//   XtsTransport/XtsTransport Instance <-> NC-Task 1/Axes/Mover Axis 105
//     PlcTask Inputs/GVL_XTS.AxisRefMover[105].NcToPlc <-> Outputs/ToPlc
//     PlcTask Outputs/GVL_XTS.AxisRefMover[105].PlcToNc <-> Inputs/FromPlc
//   XtsTransport/XtsTransport Instance <-> NC-Task 1/Axes/Mover Axis 106
//     PlcTask Inputs/GVL_XTS.AxisRefMover[106].NcToPlc <-> Outputs/ToPlc
//     PlcTask Outputs/GVL_XTS.AxisRefMover[106].PlcToNc <-> Inputs/FromPlc
//   XtsTransport/XtsTransport Instance <-> NC-Task 1/Axes/Mover Axis 107
//     PlcTask Inputs/GVL_XTS.AxisRefMover[107].NcToPlc <-> Outputs/ToPlc
//     PlcTask Outputs/GVL_XTS.AxisRefMover[107].PlcToNc <-> Inputs/FromPlc
//   XtsTransport/XtsTransport Instance <-> NC-Task 1/Axes/Mover Axis 108
//     PlcTask Inputs/GVL_XTS.AxisRefMover[108].NcToPlc <-> Outputs/ToPlc
//     PlcTask Outputs/GVL_XTS.AxisRefMover[108].PlcToNc <-> Inputs/FromPlc
//   XtsTransport/XtsTransport Instance <-> NC-Task 1/Axes/Mover Axis 11
//     PlcTask Inputs/GVL_XTS.AxisRefMover[11].NcToPlc <-> Outputs/ToPlc
//     PlcTask Outputs/GVL_XTS.AxisRefMover[11].PlcToNc <-> Inputs/FromPlc
//   XtsTransport/XtsTransport Instance <-> NC-Task 1/Axes/Mover Axis 12
//     PlcTask Inputs/GVL_XTS.AxisRefMover[12].NcToPlc <-> Outputs/ToPlc
//     PlcTask Outputs/GVL_XTS.AxisRefMover[12].PlcToNc <-> Inputs/FromPlc
//   XtsTransport/XtsTransport Instance <-> NC-Task 1/Axes/Mover Axis 13
//     PlcTask Inputs/GVL_XTS.AxisRefMover[13].NcToPlc <-> Outputs/ToPlc
//     PlcTask Outputs/GVL_XTS.AxisRefMover[13].PlcToNc <-> Inputs/FromPlc
//   XtsTransport/XtsTransport Instance <-> NC-Task 1/Axes/Mover Axis 14
//     PlcTask Inputs/GVL_XTS.AxisRefMover[14].NcToPlc <-> Outputs/ToPlc
//     PlcTask Outputs/GVL_XTS.AxisRefMover[14].PlcToNc <-> Inputs/FromPlc
//   XtsTransport/XtsTransport Instance <-> NC-Task 1/Axes/Mover Axis 15
//     PlcTask Inputs/GVL_XTS.AxisRefMover[15].NcToPlc <-> Outputs/ToPlc
//     PlcTask Outputs/GVL_XTS.AxisRefMover[15].PlcToNc <-> Inputs/FromPlc
//   XtsTransport/XtsTransport Instance <-> NC-Task 1/Axes/Mover Axis 16
//     PlcTask Inputs/GVL_XTS.AxisRefMover[16].NcToPlc <-> Outputs/ToPlc
//     PlcTask Outputs/GVL_XTS.AxisRefMover[16].PlcToNc <-> Inputs/FromPlc
//   XtsTransport/XtsTransport Instance <-> NC-Task 1/Axes/Mover Axis 17
//     PlcTask Inputs/GVL_XTS.AxisRefMover[17].NcToPlc <-> Outputs/ToPlc
//     PlcTask Outputs/GVL_XTS.AxisRefMover[17].PlcToNc <-> Inputs/FromPlc
//   XtsTransport/XtsTransport Instance <-> NC-Task 1/Axes/Mover Axis 18
//     PlcTask Inputs/GVL_XTS.AxisRefMover[18].NcToPlc <-> Outputs/ToPlc
//     PlcTask Outputs/GVL_XTS.AxisRefMover[18].PlcToNc <-> Inputs/FromPlc
//   XtsTransport/XtsTransport Instance <-> NC-Task 1/Axes/Mover Axis 19
//     PlcTask Inputs/GVL_XTS.AxisRefMover[19].NcToPlc <-> Outputs/ToPlc
//     PlcTask Outputs/GVL_XTS.AxisRefMover[19].PlcToNc <-> Inputs/FromPlc
//   XtsTransport/XtsTransport Instance <-> NC-Task 1/Axes/Mover Axis 2
//     PlcTask Inputs/GVL_XTS.AxisRefMover[2].NcToPlc <-> Outputs/ToPlc
//     PlcTask Outputs/GVL_XTS.AxisRefMover[2].PlcToNc <-> Inputs/FromPlc
//   XtsTransport/XtsTransport Instance <-> NC-Task 1/Axes/Mover Axis 20
//     PlcTask Inputs/GVL_XTS.AxisRefMover[20].NcToPlc <-> Outputs/ToPlc
//     PlcTask Outputs/GVL_XTS.AxisRefMover[20].PlcToNc <-> Inputs/FromPlc
//   XtsTransport/XtsTransport Instance <-> NC-Task 1/Axes/Mover Axis 21
//     PlcTask Inputs/GVL_XTS.AxisRefMover[21].NcToPlc <-> Outputs/ToPlc
//     PlcTask Outputs/GVL_XTS.AxisRefMover[21].PlcToNc <-> Inputs/FromPlc
//   XtsTransport/XtsTransport Instance <-> NC-Task 1/Axes/Mover Axis 22
//     PlcTask Inputs/GVL_XTS.AxisRefMover[22].NcToPlc <-> Outputs/ToPlc
//     PlcTask Outputs/GVL_XTS.AxisRefMover[22].PlcToNc <-> Inputs/FromPlc
//   XtsTransport/XtsTransport Instance <-> NC-Task 1/Axes/Mover Axis 23
//     PlcTask Inputs/GVL_XTS.AxisRefMover[23].NcToPlc <-> Outputs/ToPlc
//     PlcTask Outputs/GVL_XTS.AxisRefMover[23].PlcToNc <-> Inputs/FromPlc
//   XtsTransport/XtsTransport Instance <-> NC-Task 1/Axes/Mover Axis 24
//     PlcTask Inputs/GVL_XTS.AxisRefMover[24].NcToPlc <-> Outputs/ToPlc
//     PlcTask Outputs/GVL_XTS.AxisRefMover[24].PlcToNc <-> Inputs/FromPlc
//   XtsTransport/XtsTransport Instance <-> NC-Task 1/Axes/Mover Axis 25
//     PlcTask Inputs/GVL_XTS.AxisRefMover[25].NcToPlc <-> Outputs/ToPlc
//     PlcTask Outputs/GVL_XTS.AxisRefMover[25].PlcToNc <-> Inputs/FromPlc
//   XtsTransport/XtsTransport Instance <-> NC-Task 1/Axes/Mover Axis 26
//     PlcTask Inputs/GVL_XTS.AxisRefMover[26].NcToPlc <-> Outputs/ToPlc
//     PlcTask Outputs/GVL_XTS.AxisRefMover[26].PlcToNc <-> Inputs/FromPlc
//   XtsTransport/XtsTransport Instance <-> NC-Task 1/Axes/Mover Axis 27
//     PlcTask Inputs/GVL_XTS.AxisRefMover[27].NcToPlc <-> Outputs/ToPlc
//     PlcTask Outputs/GVL_XTS.AxisRefMover[27].PlcToNc <-> Inputs/FromPlc
//   XtsTransport/XtsTransport Instance <-> NC-Task 1/Axes/Mover Axis 28
//     PlcTask Inputs/GVL_XTS.AxisRefMover[28].NcToPlc <-> Outputs/ToPlc
//     PlcTask Outputs/GVL_XTS.AxisRefMover[28].PlcToNc <-> Inputs/FromPlc
//   XtsTransport/XtsTransport Instance <-> NC-Task 1/Axes/Mover Axis 29
//     PlcTask Inputs/GVL_XTS.AxisRefMover[29].NcToPlc <-> Outputs/ToPlc
//     PlcTask Outputs/GVL_XTS.AxisRefMover[29].PlcToNc <-> Inputs/FromPlc
//   XtsTransport/XtsTransport Instance <-> NC-Task 1/Axes/Mover Axis 3
//     PlcTask Inputs/GVL_XTS.AxisRefMover[3].NcToPlc <-> Outputs/ToPlc
//     PlcTask Outputs/GVL_XTS.AxisRefMover[3].PlcToNc <-> Inputs/FromPlc
//   XtsTransport/XtsTransport Instance <-> NC-Task 1/Axes/Mover Axis 30
//     PlcTask Inputs/GVL_XTS.AxisRefMover[30].NcToPlc <-> Outputs/ToPlc
//     PlcTask Outputs/GVL_XTS.AxisRefMover[30].PlcToNc <-> Inputs/FromPlc
//   XtsTransport/XtsTransport Instance <-> NC-Task 1/Axes/Mover Axis 31
//     PlcTask Inputs/GVL_XTS.AxisRefMover[31].NcToPlc <-> Outputs/ToPlc
//     PlcTask Outputs/GVL_XTS.AxisRefMover[31].PlcToNc <-> Inputs/FromPlc
//   XtsTransport/XtsTransport Instance <-> NC-Task 1/Axes/Mover Axis 32
//     PlcTask Inputs/GVL_XTS.AxisRefMover[32].NcToPlc <-> Outputs/ToPlc
//     PlcTask Outputs/GVL_XTS.AxisRefMover[32].PlcToNc <-> Inputs/FromPlc
//   XtsTransport/XtsTransport Instance <-> NC-Task 1/Axes/Mover Axis 33
//     PlcTask Inputs/GVL_XTS.AxisRefMover[33].NcToPlc <-> Outputs/ToPlc
//     PlcTask Outputs/GVL_XTS.AxisRefMover[33].PlcToNc <-> Inputs/FromPlc
//   XtsTransport/XtsTransport Instance <-> NC-Task 1/Axes/Mover Axis 34
//     PlcTask Inputs/GVL_XTS.AxisRefMover[34].NcToPlc <-> Outputs/ToPlc
//     PlcTask Outputs/GVL_XTS.AxisRefMover[34].PlcToNc <-> Inputs/FromPlc
//   XtsTransport/XtsTransport Instance <-> NC-Task 1/Axes/Mover Axis 35
//     PlcTask Inputs/GVL_XTS.AxisRefMover[35].NcToPlc <-> Outputs/ToPlc
//     PlcTask Outputs/GVL_XTS.AxisRefMover[35].PlcToNc <-> Inputs/FromPlc
//   XtsTransport/XtsTransport Instance <-> NC-Task 1/Axes/Mover Axis 36
//     PlcTask Inputs/GVL_XTS.AxisRefMover[36].NcToPlc <-> Outputs/ToPlc
//     PlcTask Outputs/GVL_XTS.AxisRefMover[36].PlcToNc <-> Inputs/FromPlc
//   XtsTransport/XtsTransport Instance <-> NC-Task 1/Axes/Mover Axis 37
//     PlcTask Inputs/GVL_XTS.AxisRefMover[37].NcToPlc <-> Outputs/ToPlc
//     PlcTask Outputs/GVL_XTS.AxisRefMover[37].PlcToNc <-> Inputs/FromPlc
//   XtsTransport/XtsTransport Instance <-> NC-Task 1/Axes/Mover Axis 38
//     PlcTask Inputs/GVL_XTS.AxisRefMover[38].NcToPlc <-> Outputs/ToPlc
//     PlcTask Outputs/GVL_XTS.AxisRefMover[38].PlcToNc <-> Inputs/FromPlc
//   XtsTransport/XtsTransport Instance <-> NC-Task 1/Axes/Mover Axis 39
//     PlcTask Inputs/GVL_XTS.AxisRefMover[39].NcToPlc <-> Outputs/ToPlc
//     PlcTask Outputs/GVL_XTS.AxisRefMover[39].PlcToNc <-> Inputs/FromPlc
//   XtsTransport/XtsTransport Instance <-> NC-Task 1/Axes/Mover Axis 4
//     PlcTask Inputs/GVL_XTS.AxisRefMover[4].NcToPlc <-> Outputs/ToPlc
//     PlcTask Outputs/GVL_XTS.AxisRefMover[4].PlcToNc <-> Inputs/FromPlc
//   XtsTransport/XtsTransport Instance <-> NC-Task 1/Axes/Mover Axis 40
//     PlcTask Inputs/GVL_XTS.AxisRefMover[40].NcToPlc <-> Outputs/ToPlc
//     PlcTask Outputs/GVL_XTS.AxisRefMover[40].PlcToNc <-> Inputs/FromPlc
//   XtsTransport/XtsTransport Instance <-> NC-Task 1/Axes/Mover Axis 41
//     PlcTask Inputs/GVL_XTS.AxisRefMover[41].NcToPlc <-> Outputs/ToPlc
//     PlcTask Outputs/GVL_XTS.AxisRefMover[41].PlcToNc <-> Inputs/FromPlc
//   XtsTransport/XtsTransport Instance <-> NC-Task 1/Axes/Mover Axis 42
//     PlcTask Inputs/GVL_XTS.AxisRefMover[42].NcToPlc <-> Outputs/ToPlc
//     PlcTask Outputs/GVL_XTS.AxisRefMover[42].PlcToNc <-> Inputs/FromPlc
//   XtsTransport/XtsTransport Instance <-> NC-Task 1/Axes/Mover Axis 43
//     PlcTask Inputs/GVL_XTS.AxisRefMover[43].NcToPlc <-> Outputs/ToPlc
//     PlcTask Outputs/GVL_XTS.AxisRefMover[43].PlcToNc <-> Inputs/FromPlc
//   XtsTransport/XtsTransport Instance <-> NC-Task 1/Axes/Mover Axis 44
//     PlcTask Inputs/GVL_XTS.AxisRefMover[44].NcToPlc <-> Outputs/ToPlc
//     PlcTask Outputs/GVL_XTS.AxisRefMover[44].PlcToNc <-> Inputs/FromPlc
//   XtsTransport/XtsTransport Instance <-> NC-Task 1/Axes/Mover Axis 45
//     PlcTask Inputs/GVL_XTS.AxisRefMover[45].NcToPlc <-> Outputs/ToPlc
//     PlcTask Outputs/GVL_XTS.AxisRefMover[45].PlcToNc <-> Inputs/FromPlc
//   XtsTransport/XtsTransport Instance <-> NC-Task 1/Axes/Mover Axis 46
//     PlcTask Inputs/GVL_XTS.AxisRefMover[46].NcToPlc <-> Outputs/ToPlc
//     PlcTask Outputs/GVL_XTS.AxisRefMover[46].PlcToNc <-> Inputs/FromPlc
//   XtsTransport/XtsTransport Instance <-> NC-Task 1/Axes/Mover Axis 47
//     PlcTask Inputs/GVL_XTS.AxisRefMover[47].NcToPlc <-> Outputs/ToPlc
//     PlcTask Outputs/GVL_XTS.AxisRefMover[47].PlcToNc <-> Inputs/FromPlc
//   XtsTransport/XtsTransport Instance <-> NC-Task 1/Axes/Mover Axis 48
//     PlcTask Inputs/GVL_XTS.AxisRefMover[48].NcToPlc <-> Outputs/ToPlc
//     PlcTask Outputs/GVL_XTS.AxisRefMover[48].PlcToNc <-> Inputs/FromPlc
//   XtsTransport/XtsTransport Instance <-> NC-Task 1/Axes/Mover Axis 49
//     PlcTask Inputs/GVL_XTS.AxisRefMover[49].NcToPlc <-> Outputs/ToPlc
//     PlcTask Outputs/GVL_XTS.AxisRefMover[49].PlcToNc <-> Inputs/FromPlc
//   XtsTransport/XtsTransport Instance <-> NC-Task 1/Axes/Mover Axis 5
//     PlcTask Inputs/GVL_XTS.AxisRefMover[5].NcToPlc <-> Outputs/ToPlc
//     PlcTask Outputs/GVL_XTS.AxisRefMover[5].PlcToNc <-> Inputs/FromPlc
//   XtsTransport/XtsTransport Instance <-> NC-Task 1/Axes/Mover Axis 50
//     PlcTask Inputs/GVL_XTS.AxisRefMover[50].NcToPlc <-> Outputs/ToPlc
//     PlcTask Outputs/GVL_XTS.AxisRefMover[50].PlcToNc <-> Inputs/FromPlc
//   XtsTransport/XtsTransport Instance <-> NC-Task 1/Axes/Mover Axis 51
//     PlcTask Inputs/GVL_XTS.AxisRefMover[51].NcToPlc <-> Outputs/ToPlc
//     PlcTask Outputs/GVL_XTS.AxisRefMover[51].PlcToNc <-> Inputs/FromPlc
//   XtsTransport/XtsTransport Instance <-> NC-Task 1/Axes/Mover Axis 52
//     PlcTask Inputs/GVL_XTS.AxisRefMover[52].NcToPlc <-> Outputs/ToPlc
//     PlcTask Outputs/GVL_XTS.AxisRefMover[52].PlcToNc <-> Inputs/FromPlc
//   XtsTransport/XtsTransport Instance <-> NC-Task 1/Axes/Mover Axis 53
//     PlcTask Inputs/GVL_XTS.AxisRefMover[53].NcToPlc <-> Outputs/ToPlc
//     PlcTask Outputs/GVL_XTS.AxisRefMover[53].PlcToNc <-> Inputs/FromPlc
//   XtsTransport/XtsTransport Instance <-> NC-Task 1/Axes/Mover Axis 54
//     PlcTask Inputs/GVL_XTS.AxisRefMover[54].NcToPlc <-> Outputs/ToPlc
//     PlcTask Outputs/GVL_XTS.AxisRefMover[54].PlcToNc <-> Inputs/FromPlc
//   XtsTransport/XtsTransport Instance <-> NC-Task 1/Axes/Mover Axis 55
//     PlcTask Inputs/GVL_XTS.AxisRefMover[55].NcToPlc <-> Outputs/ToPlc
//     PlcTask Outputs/GVL_XTS.AxisRefMover[55].PlcToNc <-> Inputs/FromPlc
//   XtsTransport/XtsTransport Instance <-> NC-Task 1/Axes/Mover Axis 56
//     PlcTask Inputs/GVL_XTS.AxisRefMover[56].NcToPlc <-> Outputs/ToPlc
//     PlcTask Outputs/GVL_XTS.AxisRefMover[56].PlcToNc <-> Inputs/FromPlc
//   XtsTransport/XtsTransport Instance <-> NC-Task 1/Axes/Mover Axis 57
//     PlcTask Inputs/GVL_XTS.AxisRefMover[57].NcToPlc <-> Outputs/ToPlc
//     PlcTask Outputs/GVL_XTS.AxisRefMover[57].PlcToNc <-> Inputs/FromPlc
//   XtsTransport/XtsTransport Instance <-> NC-Task 1/Axes/Mover Axis 58
//     PlcTask Inputs/GVL_XTS.AxisRefMover[58].NcToPlc <-> Outputs/ToPlc
//     PlcTask Outputs/GVL_XTS.AxisRefMover[58].PlcToNc <-> Inputs/FromPlc
//   XtsTransport/XtsTransport Instance <-> NC-Task 1/Axes/Mover Axis 59
//     PlcTask Inputs/GVL_XTS.AxisRefMover[59].NcToPlc <-> Outputs/ToPlc
//     PlcTask Outputs/GVL_XTS.AxisRefMover[59].PlcToNc <-> Inputs/FromPlc
//   XtsTransport/XtsTransport Instance <-> NC-Task 1/Axes/Mover Axis 6
//     PlcTask Inputs/GVL_XTS.AxisRefMover[6].NcToPlc <-> Outputs/ToPlc
//     PlcTask Outputs/GVL_XTS.AxisRefMover[6].PlcToNc <-> Inputs/FromPlc
//   XtsTransport/XtsTransport Instance <-> NC-Task 1/Axes/Mover Axis 60
//     PlcTask Inputs/GVL_XTS.AxisRefMover[60].NcToPlc <-> Outputs/ToPlc
//     PlcTask Outputs/GVL_XTS.AxisRefMover[60].PlcToNc <-> Inputs/FromPlc
//   XtsTransport/XtsTransport Instance <-> NC-Task 1/Axes/Mover Axis 61
//     PlcTask Inputs/GVL_XTS.AxisRefMover[61].NcToPlc <-> Outputs/ToPlc
//     PlcTask Outputs/GVL_XTS.AxisRefMover[61].PlcToNc <-> Inputs/FromPlc
//   XtsTransport/XtsTransport Instance <-> NC-Task 1/Axes/Mover Axis 62
//     PlcTask Inputs/GVL_XTS.AxisRefMover[62].NcToPlc <-> Outputs/ToPlc
//     PlcTask Outputs/GVL_XTS.AxisRefMover[62].PlcToNc <-> Inputs/FromPlc
//   XtsTransport/XtsTransport Instance <-> NC-Task 1/Axes/Mover Axis 63
//     PlcTask Inputs/GVL_XTS.AxisRefMover[63].NcToPlc <-> Outputs/ToPlc
//     PlcTask Outputs/GVL_XTS.AxisRefMover[63].PlcToNc <-> Inputs/FromPlc
//   XtsTransport/XtsTransport Instance <-> NC-Task 1/Axes/Mover Axis 64
//     PlcTask Inputs/GVL_XTS.AxisRefMover[64].NcToPlc <-> Outputs/ToPlc
//     PlcTask Outputs/GVL_XTS.AxisRefMover[64].PlcToNc <-> Inputs/FromPlc
//   XtsTransport/XtsTransport Instance <-> NC-Task 1/Axes/Mover Axis 65
//     PlcTask Inputs/GVL_XTS.AxisRefMover[65].NcToPlc <-> Outputs/ToPlc
//     PlcTask Outputs/GVL_XTS.AxisRefMover[65].PlcToNc <-> Inputs/FromPlc
//   XtsTransport/XtsTransport Instance <-> NC-Task 1/Axes/Mover Axis 66
//     PlcTask Inputs/GVL_XTS.AxisRefMover[66].NcToPlc <-> Outputs/ToPlc
//     PlcTask Outputs/GVL_XTS.AxisRefMover[66].PlcToNc <-> Inputs/FromPlc
//   XtsTransport/XtsTransport Instance <-> NC-Task 1/Axes/Mover Axis 67
//     PlcTask Inputs/GVL_XTS.AxisRefMover[67].NcToPlc <-> Outputs/ToPlc
//     PlcTask Outputs/GVL_XTS.AxisRefMover[67].PlcToNc <-> Inputs/FromPlc
//   XtsTransport/XtsTransport Instance <-> NC-Task 1/Axes/Mover Axis 68
//     PlcTask Inputs/GVL_XTS.AxisRefMover[68].NcToPlc <-> Outputs/ToPlc
//     PlcTask Outputs/GVL_XTS.AxisRefMover[68].PlcToNc <-> Inputs/FromPlc
//   XtsTransport/XtsTransport Instance <-> NC-Task 1/Axes/Mover Axis 69
//     PlcTask Inputs/GVL_XTS.AxisRefMover[69].NcToPlc <-> Outputs/ToPlc
//     PlcTask Outputs/GVL_XTS.AxisRefMover[69].PlcToNc <-> Inputs/FromPlc
//   XtsTransport/XtsTransport Instance <-> NC-Task 1/Axes/Mover Axis 7
//     PlcTask Inputs/GVL_XTS.AxisRefMover[7].NcToPlc <-> Outputs/ToPlc
//     PlcTask Outputs/GVL_XTS.AxisRefMover[7].PlcToNc <-> Inputs/FromPlc
//   XtsTransport/XtsTransport Instance <-> NC-Task 1/Axes/Mover Axis 70
//     PlcTask Inputs/GVL_XTS.AxisRefMover[70].NcToPlc <-> Outputs/ToPlc
//     PlcTask Outputs/GVL_XTS.AxisRefMover[70].PlcToNc <-> Inputs/FromPlc
//   XtsTransport/XtsTransport Instance <-> NC-Task 1/Axes/Mover Axis 71
//     PlcTask Inputs/GVL_XTS.AxisRefMover[71].NcToPlc <-> Outputs/ToPlc
//     PlcTask Outputs/GVL_XTS.AxisRefMover[71].PlcToNc <-> Inputs/FromPlc
//   XtsTransport/XtsTransport Instance <-> NC-Task 1/Axes/Mover Axis 72
//     PlcTask Inputs/GVL_XTS.AxisRefMover[72].NcToPlc <-> Outputs/ToPlc
//     PlcTask Outputs/GVL_XTS.AxisRefMover[72].PlcToNc <-> Inputs/FromPlc
//   XtsTransport/XtsTransport Instance <-> NC-Task 1/Axes/Mover Axis 73
//     PlcTask Inputs/GVL_XTS.AxisRefMover[73].NcToPlc <-> Outputs/ToPlc
//     PlcTask Outputs/GVL_XTS.AxisRefMover[73].PlcToNc <-> Inputs/FromPlc
//   XtsTransport/XtsTransport Instance <-> NC-Task 1/Axes/Mover Axis 74
//     PlcTask Inputs/GVL_XTS.AxisRefMover[74].NcToPlc <-> Outputs/ToPlc
//     PlcTask Outputs/GVL_XTS.AxisRefMover[74].PlcToNc <-> Inputs/FromPlc
//   XtsTransport/XtsTransport Instance <-> NC-Task 1/Axes/Mover Axis 75
//     PlcTask Inputs/GVL_XTS.AxisRefMover[75].NcToPlc <-> Outputs/ToPlc
//     PlcTask Outputs/GVL_XTS.AxisRefMover[75].PlcToNc <-> Inputs/FromPlc
//   XtsTransport/XtsTransport Instance <-> NC-Task 1/Axes/Mover Axis 76
//     PlcTask Inputs/GVL_XTS.AxisRefMover[76].NcToPlc <-> Outputs/ToPlc
//     PlcTask Outputs/GVL_XTS.AxisRefMover[76].PlcToNc <-> Inputs/FromPlc
//   XtsTransport/XtsTransport Instance <-> NC-Task 1/Axes/Mover Axis 77
//     PlcTask Inputs/GVL_XTS.AxisRefMover[77].NcToPlc <-> Outputs/ToPlc
//     PlcTask Outputs/GVL_XTS.AxisRefMover[77].PlcToNc <-> Inputs/FromPlc
//   XtsTransport/XtsTransport Instance <-> NC-Task 1/Axes/Mover Axis 78
//     PlcTask Inputs/GVL_XTS.AxisRefMover[78].NcToPlc <-> Outputs/ToPlc
//     PlcTask Outputs/GVL_XTS.AxisRefMover[78].PlcToNc <-> Inputs/FromPlc
//   XtsTransport/XtsTransport Instance <-> NC-Task 1/Axes/Mover Axis 79
//     PlcTask Inputs/GVL_XTS.AxisRefMover[79].NcToPlc <-> Outputs/ToPlc
//     PlcTask Outputs/GVL_XTS.AxisRefMover[79].PlcToNc <-> Inputs/FromPlc
//   XtsTransport/XtsTransport Instance <-> NC-Task 1/Axes/Mover Axis 8
//     PlcTask Inputs/GVL_XTS.AxisRefMover[8].NcToPlc <-> Outputs/ToPlc
//     PlcTask Outputs/GVL_XTS.AxisRefMover[8].PlcToNc <-> Inputs/FromPlc
//   XtsTransport/XtsTransport Instance <-> NC-Task 1/Axes/Mover Axis 80
//     PlcTask Inputs/GVL_XTS.AxisRefMover[80].NcToPlc <-> Outputs/ToPlc
//     PlcTask Outputs/GVL_XTS.AxisRefMover[80].PlcToNc <-> Inputs/FromPlc
//   XtsTransport/XtsTransport Instance <-> NC-Task 1/Axes/Mover Axis 81
//     PlcTask Inputs/GVL_XTS.AxisRefMover[81].NcToPlc <-> Outputs/ToPlc
//     PlcTask Outputs/GVL_XTS.AxisRefMover[81].PlcToNc <-> Inputs/FromPlc
//   XtsTransport/XtsTransport Instance <-> NC-Task 1/Axes/Mover Axis 82
//     PlcTask Inputs/GVL_XTS.AxisRefMover[82].NcToPlc <-> Outputs/ToPlc
//     PlcTask Outputs/GVL_XTS.AxisRefMover[82].PlcToNc <-> Inputs/FromPlc
//   XtsTransport/XtsTransport Instance <-> NC-Task 1/Axes/Mover Axis 83
//     PlcTask Inputs/GVL_XTS.AxisRefMover[83].NcToPlc <-> Outputs/ToPlc
//     PlcTask Outputs/GVL_XTS.AxisRefMover[83].PlcToNc <-> Inputs/FromPlc
//   XtsTransport/XtsTransport Instance <-> NC-Task 1/Axes/Mover Axis 84
//     PlcTask Inputs/GVL_XTS.AxisRefMover[84].NcToPlc <-> Outputs/ToPlc
//     PlcTask Outputs/GVL_XTS.AxisRefMover[84].PlcToNc <-> Inputs/FromPlc
//   XtsTransport/XtsTransport Instance <-> NC-Task 1/Axes/Mover Axis 85
//     PlcTask Inputs/GVL_XTS.AxisRefMover[85].NcToPlc <-> Outputs/ToPlc
//     PlcTask Outputs/GVL_XTS.AxisRefMover[85].PlcToNc <-> Inputs/FromPlc
